LIN {X 0,Y 270.05,Z 181.094,A -85,B 0,C 180,E1 -19060.447,E2 -19060.447} C_VEL
LIN {X 0,Y 266.904,Z 176.821,A -85,B 0,C 180,E1 -19061.814,E2 -19061.814} C_VEL
LIN {X 0,Y 264.347,Z 175.041,A -85,B 0,C 180,E1 -19062.905,E2 -19062.905} C_VEL
LIN {X 0,Y 256.649,Z 172.883,A -85,B 0,C 180,E1 -19066.441,E2 -19066.441} C_VEL
LIN {X 0,Y 254.506,Z 171.313,A -85,B 0,C 180,E1 -19067.626,E2 -19067.626} C_VEL
LIN {X 0,Y 253.888,Z 170.514,A -85,B 0,C 180,E1 -19068.008,E2 -19068.008} C_VEL
LIN {X 0,Y 252.108,Z 167.577,A -85,B 0,C 180,E1 -19069.204,E2 -19069.204} C_VEL
LIN {X 0,Y 249.588,Z 165.512,A -85,B 0,C 180,E1 -19070.909,E2 -19070.909} C_VEL
LIN {X 0,Y 247.997,Z 162.813,A -85,B 0,C 180,E1 -19072.212,E2 -19072.212} C_VEL
LIN {X 0,Y 247.745,Z 162.046,A -85,B 0,C 180,E1 -19072.46,E2 -19072.46} C_VEL
LIN {X 0,Y 244.192,Z 159.968,A -85,B 0,C 180,E1 -19075.46,E2 -19075.46} C_VEL
LIN {X 0,Y 242.872,Z 157.671,A -85,B 0,C 180,E1 -19076.993,E2 -19076.993} C_VEL
LIN {X 0,Y 242.522,Z 155.89,A -85,B 0,C 180,E1 -19077.716,E2 -19077.716} C_VEL
LIN {X 0,Y 242.691,Z 155.88,A -85,B 0,C 180,E1 -19079.999,E2 -19079.999} C_VEL
LIN {X 0,Y 242.635,Z 155.875,A -85,B 0,C 180,E1 -19081.659,E2 -19081.659} C_VEL
LIN {X 0,Y 242.4,Z 155.913,A -85,B 0,C 180,E1 -19086.659,E2 -19086.659} C_VEL
LIN {X 0,Y 242.265,Z 155.926,A -85,B 0,C 180,E1 -19090.023,E2 -19090.023} C_VEL
LIN {X 0,Y 242.166,Z 155.938,A -85,B 0,C 180,E1 -19095.14,E2 -19095.14} C_VEL
LIN {X 0,Y 242.075,Z 155.945,A -85,B 0,C 180,E1 -19099.669,E2 -19099.669} C_VEL
LIN {X 0,Y 242.299,Z 157.093,A -85,B 0,C 180,E1 -19100.991,E2 -19100.991} C_VEL
LIN {X 0,Y 243.437,Z 159.421,A -85,B 0,C 180,E1 -19102.448,E2 -19102.448} C_VEL
LIN {X 0,Y 246.039,Z 161.798,A -85,B 0,C 180,E1 -19104.918,E2 -19104.918} C_VEL
LIN {X 0,Y 248.946,Z 165.199,A -85,B 0,C 180,E1 -19107.306,E2 -19107.306} C_VEL
LIN {X 0,Y 252.346,Z 169.692,A -85,B 0,C 180,E1 -19109.752,E2 -19109.752} C_VEL
LIN {X 0,Y 253.782,Z 171.342,A -85,B 0,C 180,E1 -19110.657,E2 -19110.657} C_VEL
LIN {X 0,Y 258.589,Z 177.663,A -85,B 0,C 180,E1 -19113.449,E2 -19113.449} C_VEL
LIN {X 0,Y 262.502,Z 183.277,A -85,B 0,C 180,E1 -19115.489,E2 -19115.489} C_VEL
LIN {X 0,Y 268.007,Z 191.52,A -85,B 0,C 180,E1 -19118.035,E2 -19118.035} C_VEL
LIN {X 0,Y 273.834,Z 200.761,A -85,B 0,C 180,E1 -19120.447,E2 -19120.447} C_VEL
LIN {X 0,Y 279.53,Z 210.74,A -85,B 0,C 180,E1 -19122.615,E2 -19122.615} C_VEL
LIN {X 0,Y 285.287,Z 221.644,A -85,B 0,C 180,E1 -19124.619,E2 -19124.619} C_VEL
LIN {X 0,Y 291.028,Z 234.204,A -85,B 0,C 180,E1 -19126.505,E2 -19126.505} C_VEL
LIN {X 0,Y 291.336,Z 235.609,A -85,B 0,C 180,E1 -19126.631,E2 -19126.631} C_VEL
LIN {X 0,Y 285.753,Z 326.096,A -85,B 0,C 180,E1 -19128.86,E2 -19128.86} C_VEL
LIN {X 0,Y 283.787,Z 341.992,A -85,B 0,C 180,E1 -19129.453,E2 -19129.453} C_VEL
LIN {X 0,Y 281.088,Z 357.105,A -85,B 0,C 180,E1 -19130.273,E2 -19130.273} C_VEL
LIN {X 0,Y 278.009,Z 370.686,A -85,B 0,C 180,E1 -19131.269,E2 -19131.269} C_VEL
LIN {X 0,Y 274.119,Z 385.222,A -85,B 0,C 180,E1 -19132.661,E2 -19132.661} C_VEL
LIN {X 0,Y 270.67,Z 396.438,A -85,B 0,C 180,E1 -19134.023,E2 -19134.023} C_VEL
LIN {X 0,Y 266.245,Z 409.051,A -85,B 0,C 180,E1 -19135.88,E2 -19135.88} C_VEL
LIN {X 0,Y 261.748,Z 420.548,A -85,B 0,C 180,E1 -19137.975,E2 -19137.975} C_VEL
LIN {X 0,Y 257.041,Z 431.736,A -85,B 0,C 180,E1 -19140.518,E2 -19140.518} C_VEL
LIN {X 0,Y 253.709,Z 439.245,A -85,B 0,C 180,E1 -19142.582,E2 -19142.582} C_VEL
LIN {X 0,Y 249.879,Z 447.882,A -85,B 0,C 180,E1 -19145.491,E2 -19145.491} C_VEL
LIN {X 0,Y 246.86,Z 454.558,A -85,B 0,C 180,E1 -19148.279,E2 -19148.279} C_VEL
LIN {X 0,Y 244,Z 460.761,A -85,B 0,C 180,E1 -19151.529,E2 -19151.529} C_VEL
LIN {X 0,Y 242.026,Z 465.605,A -85,B 0,C 180,E1 -19154.851,E2 -19154.851} C_VEL
LIN {X 0,Y 240.671,Z 469.21,A -85,B 0,C 180,E1 -19158.206,E2 -19158.206} C_VEL
LIN {X 0,Y 239.979,Z 471.652,A -85,B 0,C 180,E1 -19161.581,E2 -19161.581} C_VEL
LIN {X 0,Y 239.733,Z 473.016,A -85,B 0,C 180,E1 -19165.368,E2 -19165.368} C_VEL
LIN {X 0,Y 239.826,Z 473.079,A -85,B 0,C 180,E1 -19168.321,E2 -19168.321} C_VEL
LIN {X 0,Y 239.912,Z 472.714,A -85,B 0,C 180,E1 -19170.001,E2 -19170.001} C_VEL
LIN {X 0,Y 239.783,Z 471.099,A -85,B 0,C 180,E1 -19173.361,E2 -19173.361} C_VEL
LIN {X 0,Y 239.876,Z 468.281,A -85,B 0,C 180,E1 -19176.731,E2 -19176.731} C_VEL
LIN {X 0,Y 240.194,Z 464.175,A -85,B 0,C 180,E1 -19180.112,E2 -19180.112} C_VEL
LIN {X 0,Y 241.031,Z 458.673,A -85,B 0,C 180,E1 -19183.49,E2 -19183.49} C_VEL
LIN {X 0,Y 242.441,Z 451.405,A -85,B 0,C 180,E1 -19186.94,E2 -19186.94} C_VEL
LIN {X 0,Y 244.164,Z 444.018,A -85,B 0,C 180,E1 -19189.769,E2 -19189.769} C_VEL
LIN {X 0,Y 246.564,Z 434.858,A -85,B 0,C 180,E1 -19192.632,E2 -19192.632} C_VEL
LIN {X 0,Y 249.211,Z 424.133,A -85,B 0,C 180,E1 -19195.381,E2 -19195.381} C_VEL
LIN {X 0,Y 252.238,Z 412.368,A -85,B 0,C 180,E1 -19197.821,E2 -19197.821} C_VEL
LIN {X 0,Y 255.134,Z 399.787,A -85,B 0,C 180,E1 -19199.953,E2 -19199.953} C_VEL
LIN {X 0,Y 257.953,Z 387.419,A -85,B 0,C 180,E1 -19201.634,E2 -19201.634} C_VEL
LIN {X 0,Y 260.774,Z 372.915,A -85,B 0,C 180,E1 -19203.222,E2 -19203.222} C_VEL
LIN {X 0,Y 263.081,Z 358.225,A -85,B 0,C 180,E1 -19204.473,E2 -19204.473} C_VEL
LIN {X 0,Y 265.181,Z 342.628,A -85,B 0,C 180,E1 -19205.434,E2 -19205.434} C_VEL
LIN {X 0,Y 266.583,Z 327.14,A -85,B 0,C 180,E1 -19206.091,E2 -19206.091} C_VEL
LIN {X 0,Y 271.19,Z 222.807,A -85,B 0,C 180,E1 -19208.824,E2 -19208.824} C_VEL
LIN {X 0,Y 270.291,Z 218.299,A -85,B 0,C 180,E1 -19209.091,E2 -19209.091} C_VEL
LIN {X 0,Y 263.458,Z 201.272,A -85,B 0,C 180,E1 -19210.628,E2 -19210.628} C_VEL
LIN {X 0,Y 255.801,Z 184.265,A -85,B 0,C 180,E1 -19212.402,E2 -19212.402} C_VEL
LIN {X 0,Y 248.125,Z 169.408,A -85,B 0,C 180,E1 -19214.242,E2 -19214.242} C_VEL
LIN {X 0,Y 243.223,Z 160.405,A -85,B 0,C 180,E1 -19215.517,E2 -19215.517} C_VEL
LIN {X 0,Y 241.97,Z 155.973,A -85,B 0,C 180,E1 -19217.349,E2 -19217.349} C_VEL
LIN {X 0,Y 241.997,Z 155.954,A -85,B 0,C 180,E1 -19221.641,E2 -19221.641} C_VEL
LIN {X 0,Y 241.989,Z 155.963,A -85,B 0,C 180,E1 -19224.49,E2 -19224.49} C_VEL
LIN {X 0,Y 241.955,Z 155.97,A -85,B 0,C 180,E1 -19228.478,E2 -19228.478} C_VEL
LIN {X 0,Y 241.97,Z 155.934,A -85,B 0,C 180,E1 -19232.309,E2 -19232.309} C_VEL
LIN {X 0,Y 242.028,Z 155.96,A -85,B 0,C 180,E1 -19236.014,E2 -19236.014} C_VEL
LIN {X 0,Y 242.025,Z 155.958,A -85,B 0,C 180,E1 -19239.607,E2 -19239.607} C_VEL
LIN {X 0,Y 242.131,Z 155.938,A -85,B 0,C 180,E1 -19243.308,E2 -19243.308} C_VEL
LIN {X 0,Y 242.172,Z 155.936,A -85,B 0,C 180,E1 -19248.28,E2 -19248.28} C_VEL
LIN {X 0,Y 242.376,Z 155.912,A -85,B 0,C 180,E1 -19251.664,E2 -19251.664} C_VEL
LIN {X 0,Y 242.401,Z 155.911,A -85,B 0,C 180,E1 -19253.341,E2 -19253.341} C_VEL
LIN {X 0,Y 242.621,Z 155.851,A -85,B 0,C 180,E1 -19258.341,E2 -19258.341} C_VEL
LIN {X 0,Y 242.619,Z 155.864,A -85,B 0,C 180,E1 -19261.661,E2 -19261.661} C_VEL
LIN {X 0,Y 242.4,Z 155.901,A -85,B 0,C 180,E1 -19266.66,E2 -19266.66} C_VEL
LIN {X 0,Y 242.264,Z 155.888,A -85,B 0,C 180,E1 -19270.025,E2 -19270.025} C_VEL
LIN {X 0,Y 242.106,Z 155.951,A -85,B 0,C 180,E1 -19275.145,E2 -19275.145} C_VEL
LIN {X 0,Y 242.013,Z 155.961,A -85,B 0,C 180,E1 -19278.63,E2 -19278.63} C_VEL
LIN {X 0,Y 241.975,Z 155.958,A -85,B 0,C 180,E1 -19282.184,E2 -19282.184} C_VEL
LIN {X 0,Y 241.991,Z 155.962,A -85,B 0,C 180,E1 -19285.827,E2 -19285.827} C_VEL
LIN {X 0,Y 241.967,Z 155.928,A -85,B 0,C 180,E1 -19289.59,E2 -19289.59} C_VEL
LIN {X 0,Y 241.983,Z 155.967,A -85,B 0,C 180,E1 -19293.493,E2 -19293.493} C_VEL
LIN {X 0,Y 241.988,Z 155.932,A -85,B 0,C 180,E1 -19297.583,E2 -19297.583} C_VEL
LIN {X 0,Y 241.923,Z 155.974,A -85,B 0,C 180,E1 -19301.927,E2 -19301.927} C_VEL
LIN {X 0,Y 241.904,Z 155.951,A -85,B 0,C 180,E1 -19306.58,E2 -19306.58} C_VEL
LIN {X 0,Y 241.934,Z 155.969,A -85,B 0,C 180,E1 -19310.276,E2 -19310.276} C_VEL
LIN {X 0,Y 241.978,Z 155.966,A -85,B 0,C 180,E1 -19314.487,E2 -19314.487} C_VEL
LIN {X 0,Y 241.958,Z 155.961,A -85,B 0,C 180,E1 -19318.476,E2 -19318.476} C_VEL
LIN {X 0,Y 241.969,Z 155.963,A -85,B 0,C 180,E1 -19322.307,E2 -19322.307} C_VEL
LIN {X 0,Y 241.999,Z 156.029,A -85,B 0,C 180,E1 -19323.589,E2 -19323.589} C_VEL
LIN {X 0,Y 242.921,Z 158.683,A -85,B 0,C 180,E1 -19323.869,E2 -19323.869} C_VEL
LIN {X 0,Y 244.718,Z 161.076,A -85,B 0,C 180,E1 -19324.3,E2 -19324.3} C_VEL
LIN {X 0,Y 256.472,Z 180.366,A -85,B 0,C 180,E1 -19327.043,E2 -19327.043} C_VEL
LIN {X 0,Y 262.923,Z 192.515,A -85,B 0,C 180,E1 -19328.47,E2 -19328.47} C_VEL
LIN {X 0,Y 269.632,Z 208.086,A -85,B 0,C 180,E1 -19329.962,E2 -19329.962} C_VEL
LIN {X 0,Y 271.569,Z 213.034,A -85,B 0,C 180,E1 -19330.389,E2 -19330.389} C_VEL
LIN {X 0,Y 266.876,Z 314.239,A -85,B 0,C 180,E1 -19333.013,E2 -19333.013} C_VEL
LIN {X 0,Y 265.518,Z 330.347,A -85,B 0,C 180,E1 -19333.715,E2 -19333.715} C_VEL
LIN {X 0,Y 263.826,Z 344.934,A -85,B 0,C 180,E1 -19334.649,E2 -19334.649} C_VEL
LIN {X 0,Y 261.727,Z 358.741,A -85,B 0,C 180,E1 -19335.816,E2 -19335.816} C_VEL
LIN {X 0,Y 259.363,Z 371.908,A -85,B 0,C 180,E1 -19337.229,E2 -19337.229} C_VEL
LIN {X 0,Y 256.641,Z 384.864,A -85,B 0,C 180,E1 -19338.948,E2 -19338.948} C_VEL
LIN {X 0,Y 253.902,Z 396.522,A -85,B 0,C 180,E1 -19340.841,E2 -19340.841} C_VEL
LIN {X 0,Y 251.026,Z 408.225,A -85,B 0,C 180,E1 -19343.166,E2 -19343.166} C_VEL
LIN {X 0,Y 248.456,Z 418.09,A -85,B 0,C 180,E1 -19345.538,E2 -19345.538} C_VEL
LIN {X 0,Y 246.001,Z 427.734,A -85,B 0,C 180,E1 -19348.362,E2 -19348.362} C_VEL
LIN {X 0,Y 243.924,Z 435.785,A -85,B 0,C 180,E1 -19351.238,E2 -19351.238} C_VEL
LIN {X 0,Y 242.335,Z 442.479,A -85,B 0,C 180,E1 -19354.157,E2 -19354.157} C_VEL
LIN {X 0,Y 241.036,Z 448.623,A -85,B 0,C 180,E1 -19357.533,E2 -19357.533} C_VEL
LIN {X 0,Y 240.172,Z 453.365,A -85,B 0,C 180,E1 -19360.964,E2 -19360.964} C_VEL
LIN {X 0,Y 239.642,Z 456.898,A -85,B 0,C 180,E1 -19364.578,E2 -19364.578} C_VEL
LIN {X 0,Y 239.493,Z 458.496,A -85,B 0,C 180,E1 -19367.064,E2 -19367.064} C_VEL
LIN {X 0,Y 239.492,Z 459.74,A -85,B 0,C 180,E1 -19370.618,E2 -19370.618} C_VEL
LIN {X 0,Y 239.842,Z 459.722,A -85,B 0,C 180,E1 -19374.219,E2 -19374.219} C_VEL
LIN {X 0,Y 240.587,Z 458.394,A -85,B 0,C 180,E1 -19377.864,E2 -19377.864} C_VEL
LIN {X 0,Y 241.902,Z 455.693,A -85,B 0,C 180,E1 -19381.53,E2 -19381.53} C_VEL
LIN {X 0,Y 243.937,Z 451.533,A -85,B 0,C 180,E1 -19385.184,E2 -19385.184} C_VEL
LIN {X 0,Y 246.746,Z 445.781,A -85,B 0,C 180,E1 -19388.801,E2 -19388.801} C_VEL
LIN {X 0,Y 249.894,Z 439.307,A -85,B 0,C 180,E1 -19391.908,E2 -19391.908} C_VEL
LIN {X 0,Y 253.681,Z 431.274,A -85,B 0,C 180,E1 -19394.946,E2 -19394.946} C_VEL
LIN {X 0,Y 258.142,Z 421.415,A -85,B 0,C 180,E1 -19397.892,E2 -19397.892} C_VEL
LIN {X 0,Y 262.699,Z 410.7,A -85,B 0,C 180,E1 -19400.441,E2 -19400.441} C_VEL
LIN {X 0,Y 267.081,Z 399.355,A -85,B 0,C 180,E1 -19402.624,E2 -19402.624} C_VEL
LIN {X 0,Y 271.14,Z 387.871,A -85,B 0,C 180,E1 -19404.414,E2 -19404.414} C_VEL
LIN {X 0,Y 275.252,Z 374.612,A -85,B 0,C 180,E1 -19406.081,E2 -19406.081} C_VEL
LIN {X 0,Y 278.751,Z 360.969,A -85,B 0,C 180,E1 -19407.462,E2 -19407.462} C_VEL
LIN {X 0,Y 282.029,Z 345.738,A -85,B 0,C 180,E1 -19408.632,E2 -19408.632} C_VEL
LIN {X 0,Y 284.295,Z 332.001,A -85,B 0,C 180,E1 -19409.426,E2 -19409.426} C_VEL
LIN {X 0,Y 286.217,Z 316.146,A -85,B 0,C 180,E1 -19410.059,E2 -19410.059} C_VEL
LIN {X 0,Y 291.678,Z 227.342,A -85,B 0,C 180,E1 -19412.267,E2 -19412.267} C_VEL
LIN {X 0,Y 286.52,Z 216.955,A -85,B 0,C 180,E1 -19413.922,E2 -19413.922} C_VEL
LIN {X 0,Y 280.857,Z 206.853,A -85,B 0,C 180,E1 -19415.843,E2 -19415.843} C_VEL
LIN {X 0,Y 276.3,Z 199.31,A -85,B 0,C 180,E1 -19417.519,E2 -19417.519} C_VEL
LIN {X 0,Y 270.649,Z 191.335,A -85,B 0,C 180,E1 -19419.718,E2 -19419.718} C_VEL
LIN {X 0,Y 267.391,Z 187.043,A -85,B 0,C 180,E1 -19421.082,E2 -19421.082} C_VEL
LIN {X 0,Y 264.021,Z 182.609,A -85,B 0,C 180,E1 -19422.595,E2 -19422.595} C_VEL
LIN {X 0,Y 261.176,Z 178.839,A -85,B 0,C 180,E1 -19423.994,E2 -19423.994} C_VEL
LIN {X 0,Y 257.612,Z 174.63,A -85,B 0,C 180,E1 -19425.862,E2 -19425.862} C_VEL
LIN {X 0,Y 256.541,Z 173.01,A -85,B 0,C 180,E1 -19426.483,E2 -19426.483} C_VEL
LIN {X 0,Y 253.888,Z 170.514,A -85,B 0,C 180,E1 -19428.008,E2 -19428.008} C_VEL
LIN {X 0,Y 251.988,Z 168.678,A -85,B 0,C 180,E1 -19429.196,E2 -19429.196} C_VEL
LIN {X 0,Y 249.958,Z 168.052,A -85,B 0,C 180,E1 -19430.459,E2 -19430.459} C_VEL
LIN {X 0,Y 244.872,Z 168.118,A -85,B 0,C 180,E1 -19434,E2 -19434} C_VEL
LIN {X 0,Y 243.834,Z 167.609,A -85,B 0,C 180,E1 -19434.905,E2 -19434.905} C_VEL
LIN {X 0,Y 241.974,Z 165.418,A -85,B 0,C 180,E1 -19436.878,E2 -19436.878} C_VEL
LIN {X 0,Y 240.963,Z 162.777,A -85,B 0,C 180,E1 -19438.328,E2 -19438.328} C_VEL
LIN {X 0,Y 236.581,Z 159.994,A -85,B 0,C 180,E1 -19448.541,E2 -19448.541} C_VEL
LIN {X 0,Y 237.634,Z 161.379,A -85,B 0,C 180,E1 -19454.997,E2 -19454.997} C_VEL
LIN {X 0,Y 240.519,Z 163.072,A -85,B 0,C 180,E1 -19459.857,E2 -19459.857} C_VEL
LIN {X 0,Y 241.092,Z 164.194,A -85,B 0,C 180,E1 -19460.684,E2 -19460.684} C_VEL
LIN {X 0,Y 242.46,Z 166.569,A -85,B 0,C 180,E1 -19462.408,E2 -19462.408} C_VEL
LIN {X 0,Y 244.723,Z 168.674,A -85,B 0,C 180,E1 -19464.604,E2 -19464.604} C_VEL
LIN {X 0,Y 247.713,Z 172.251,A -85,B 0,C 180,E1 -19467.118,E2 -19467.118} C_VEL
LIN {X 0,Y 250.494,Z 176.134,A -85,B 0,C 180,E1 -19469.197,E2 -19469.197} C_VEL
LIN {X 0,Y 251.866,Z 177.723,A -85,B 0,C 180,E1 -19470.094,E2 -19470.094} C_VEL
LIN {X 0,Y 257.149,Z 185.048,A -85,B 0,C 180,E1 -19473.266,E2 -19473.266} C_VEL
LIN {X 0,Y 261.114,Z 190.954,A -85,B 0,C 180,E1 -19475.371,E2 -19475.371} C_VEL
LIN {X 0,Y 265.433,Z 197.515,A -85,B 0,C 180,E1 -19477.424,E2 -19477.424} C_VEL
LIN {X 0,Y 271.29,Z 207.09,A -85,B 0,C 180,E1 -19479.938,E2 -19479.938} C_VEL
LIN {X 0,Y 277.493,Z 218.235,A -85,B 0,C 180,E1 -19482.363,E2 -19482.363} C_VEL
LIN {X 0,Y 282.654,Z 228.654,A -85,B 0,C 180,E1 -19484.231,E2 -19484.231} C_VEL
LIN {X 0,Y 286.593,Z 237.467,A -85,B 0,C 180,E1 -19485.579,E2 -19485.579} C_VEL
LIN {X 0,Y 280.938,Z 326.652,A -85,B 0,C 180,E1 -19487.815,E2 -19487.815} C_VEL
LIN {X 0,Y 278.906,Z 342.252,A -85,B 0,C 180,E1 -19488.409,E2 -19488.409} C_VEL
LIN {X 0,Y 275.999,Z 357.801,A -85,B 0,C 180,E1 -19489.269,E2 -19489.269} C_VEL
LIN {X 0,Y 273.075,Z 370.282,A -85,B 0,C 180,E1 -19490.194,E2 -19490.194} C_VEL
LIN {X 0,Y 268.999,Z 385.006,A -85,B 0,C 180,E1 -19491.609,E2 -19491.609} C_VEL
LIN {X 0,Y 265.419,Z 396.114,A -85,B 0,C 180,E1 -19492.959,E2 -19492.959} C_VEL
LIN {X 0,Y 260.837,Z 408.746,A -85,B 0,C 180,E1 -19494.836,E2 -19494.836} C_VEL
LIN {X 0,Y 256.529,Z 419.379,A -85,B 0,C 180,E1 -19496.775,E2 -19496.775} C_VEL
LIN {X 0,Y 252.236,Z 429.258,A -85,B 0,C 180,E1 -19498.972,E2 -19498.972} C_VEL
LIN {X 0,Y 247.788,Z 438.738,A -85,B 0,C 180,E1 -19501.551,E2 -19501.551} C_VEL
LIN {X 0,Y 243.972,Z 447.08,A -85,B 0,C 180,E1 -19504.4,E2 -19504.4} C_VEL
LIN {X 0,Y 240.238,Z 454.728,A -85,B 0,C 180,E1 -19507.648,E2 -19507.648} C_VEL
LIN {X 0,Y 237.243,Z 460.853,A -85,B 0,C 180,E1 -19510.983,E2 -19510.983} C_VEL
LIN {X 0,Y 235.103,Z 465.624,A -85,B 0,C 180,E1 -19514.393,E2 -19514.393} C_VEL
LIN {X 0,Y 233.667,Z 469.158,A -85,B 0,C 180,E1 -19517.847,E2 -19517.847} C_VEL
LIN {X 0,Y 232.918,Z 471.531,A -85,B 0,C 180,E1 -19521.323,E2 -19521.323} C_VEL
LIN {X 0,Y 232.644,Z 472.783,A -85,B 0,C 180,E1 -19524.801,E2 -19524.801} C_VEL
LIN {X 0,Y 232.737,Z 472.864,A -85,B 0,C 180,E1 -19528.27,E2 -19528.27} C_VEL
LIN {X 0,Y 232.821,Z 472.468,A -85,B 0,C 180,E1 -19530.001,E2 -19530.001} C_VEL
LIN {X 0,Y 232.693,Z 470.79,A -85,B 0,C 180,E1 -19533.464,E2 -19533.464} C_VEL
LIN {X 0,Y 232.792,Z 467.905,A -85,B 0,C 180,E1 -19536.937,E2 -19536.937} C_VEL
LIN {X 0,Y 233.139,Z 463.729,A -85,B 0,C 180,E1 -19540.421,E2 -19540.421} C_VEL
LIN {X 0,Y 234.062,Z 458.154,A -85,B 0,C 180,E1 -19543.9,E2 -19543.9} C_VEL
LIN {X 0,Y 235.539,Z 451.013,A -85,B 0,C 180,E1 -19547.361,E2 -19547.361} C_VEL
LIN {X 0,Y 237.393,Z 443.346,A -85,B 0,C 180,E1 -19550.357,E2 -19550.357} C_VEL
LIN {X 0,Y 239.93,Z 434.093,A -85,B 0,C 180,E1 -19553.294,E2 -19553.294} C_VEL
LIN {X 0,Y 242.816,Z 422.819,A -85,B 0,C 180,E1 -19556.201,E2 -19556.201} C_VEL
LIN {X 0,Y 245.869,Z 411.284,A -85,B 0,C 180,E1 -19558.607,E2 -19558.607} C_VEL
LIN {X 0,Y 248.916,Z 398.506,A -85,B 0,C 180,E1 -19560.781,E2 -19560.781} C_VEL
LIN {X 0,Y 251.821,Z 385.956,A -85,B 0,C 180,E1 -19562.497,E2 -19562.497} C_VEL
LIN {X 0,Y 254.454,Z 372.935,A -85,B 0,C 180,E1 -19563.931,E2 -19563.931} C_VEL
LIN {X 0,Y 256.812,Z 358.412,A -85,B 0,C 180,E1 -19565.199,E2 -19565.199} C_VEL
LIN {X 0,Y 258.974,Z 342.993,A -85,B 0,C 180,E1 -19566.176,E2 -19566.176} C_VEL
LIN {X 0,Y 260.407,Z 327.797,A -85,B 0,C 180,E1 -19566.846,E2 -19566.846} C_VEL
LIN {X 0,Y 265.233,Z 224.118,A -85,B 0,C 180,E1 -19569.612,E2 -19569.612} C_VEL
LIN {X 0,Y 264.413,Z 220.374,A -85,B 0,C 180,E1 -19569.853,E2 -19569.853} C_VEL
LIN {X 0,Y 256.732,Z 201.426,A -85,B 0,C 180,E1 -19571.658,E2 -19571.658} C_VEL
LIN {X 0,Y 249.37,Z 185.374,A -85,B 0,C 180,E1 -19573.436,E2 -19573.436} C_VEL
LIN {X 0,Y 242.22,Z 171.766,A -85,B 0,C 180,E1 -19575.234,E2 -19575.234} C_VEL
LIN {X 0,Y 235.916,Z 160.21,A -85,B 0,C 180,E1 -19576.945,E2 -19576.945} C_VEL
LIN {X 0,Y 234.882,Z 156.856,A -85,B 0,C 180,E1 -19578.422,E2 -19578.422} C_VEL
LIN {X 0,Y 234.92,Z 156.834,A -85,B 0,C 180,E1 -19581.08,E2 -19581.08} C_VEL
LIN {X 0,Y 234.932,Z 156.845,A -85,B 0,C 180,E1 -19585.363,E2 -19585.363} C_VEL
LIN {X 0,Y 234.901,Z 156.847,A -85,B 0,C 180,E1 -19589.429,E2 -19589.429} C_VEL
LIN {X 0,Y 234.971,Z 156.814,A -85,B 0,C 180,E1 -19593.808,E2 -19593.808} C_VEL
LIN {X 0,Y 234.993,Z 156.828,A -85,B 0,C 180,E1 -19598.969,E2 -19598.969} C_VEL
LIN {X 0,Y 235.067,Z 156.818,A -85,B 0,C 180,E1 -19603.087,E2 -19603.087} C_VEL
LIN {X 0,Y 235.104,Z 156.815,A -85,B 0,C 180,E1 -19607.922,E2 -19607.922} C_VEL
LIN {X 0,Y 235.315,Z 156.793,A -85,B 0,C 180,E1 -19611.412,E2 -19611.412} C_VEL
LIN {X 0,Y 235.352,Z 156.787,A -85,B 0,C 180,E1 -19613.141,E2 -19613.141} C_VEL
LIN {X 0,Y 235.58,Z 156.727,A -85,B 0,C 180,E1 -19618.291,E2 -19618.291} C_VEL
LIN {X 0,Y 235.578,Z 156.741,A -85,B 0,C 180,E1 -19621.71,E2 -19621.71} C_VEL
LIN {X 0,Y 235.351,Z 156.774,A -85,B 0,C 180,E1 -19626.861,E2 -19626.861} C_VEL
LIN {X 0,Y 235.187,Z 156.77,A -85,B 0,C 180,E1 -19630.329,E2 -19630.329} C_VEL
LIN {X 0,Y 235.044,Z 156.827,A -85,B 0,C 180,E1 -19635.612,E2 -19635.612} C_VEL
LIN {X 0,Y 234.956,Z 156.841,A -85,B 0,C 180,E1 -19639.211,E2 -19639.211} C_VEL
LIN {X 0,Y 234.919,Z 156.839,A -85,B 0,C 180,E1 -19642.888,E2 -19642.888} C_VEL
LIN {X 0,Y 234.926,Z 156.832,A -85,B 0,C 180,E1 -19646.664,E2 -19646.664} C_VEL
LIN {X 0,Y 234.899,Z 156.813,A -85,B 0,C 180,E1 -19650.573,E2 -19650.573} C_VEL
LIN {X 0,Y 234.927,Z 156.845,A -85,B 0,C 180,E1 -19654.639,E2 -19654.639} C_VEL
LIN {X 0,Y 234.917,Z 156.813,A -85,B 0,C 180,E1 -19658.935,E2 -19658.935} C_VEL
LIN {X 0,Y 234.866,Z 156.848,A -85,B 0,C 180,E1 -19663.492,E2 -19663.492} C_VEL
LIN {X 0,Y 234.857,Z 156.828,A -85,B 0,C 180,E1 -19666.506,E2 -19666.506} C_VEL
LIN {X 0,Y 234.923,Z 156.833,A -85,B 0,C 180,E1 -19671.078,E2 -19671.078} C_VEL
LIN {X 0,Y 234.927,Z 156.847,A -85,B 0,C 180,E1 -19675.36,E2 -19675.36} C_VEL
LIN {X 0,Y 234.904,Z 156.853,A -85,B 0,C 180,E1 -19679.427,E2 -19679.427} C_VEL
LIN {X 0,Y 234.937,Z 156.838,A -85,B 0,C 180,E1 -19682.195,E2 -19682.195} C_VEL
LIN {X 0,Y 235.938,Z 159.689,A -85,B 0,C 180,E1 -19682.53,E2 -19682.53} C_VEL
LIN {X 0,Y 237.799,Z 162.132,A -85,B 0,C 180,E1 -19683.003,E2 -19683.003} C_VEL
LIN {X 0,Y 246.976,Z 176.903,A -85,B 0,C 180,E1 -19685.309,E2 -19685.309} C_VEL
LIN {X 0,Y 254.136,Z 189.258,A -85,B 0,C 180,E1 -19686.979,E2 -19686.979} C_VEL
LIN {X 0,Y 258.788,Z 198.574,A -85,B 0,C 180,E1 -19688.04,E2 -19688.04} C_VEL
LIN {X 0,Y 265.578,Z 214.964,A -85,B 0,C 180,E1 -19689.609,E2 -19689.609} C_VEL
LIN {X 0,Y 260.744,Z 314.885,A -85,B 0,C 180,E1 -19692.246,E2 -19692.246} C_VEL
LIN {X 0,Y 259.332,Z 330.805,A -85,B 0,C 180,E1 -19692.96,E2 -19692.96} C_VEL
LIN {X 0,Y 257.524,Z 345.902,A -85,B 0,C 180,E1 -19693.959,E2 -19693.959} C_VEL
LIN {X 0,Y 255.157,Z 360.523,A -85,B 0,C 180,E1 -19695.239,E2 -19695.239} C_VEL
LIN {X 0,Y 252.495,Z 374.776,A -85,B 0,C 180,E1 -19696.861,E2 -19696.861} C_VEL
LIN {X 0,Y 249.667,Z 387.4,A -85,B 0,C 180,E1 -19698.635,E2 -19698.635} C_VEL
LIN {X 0,Y 246.618,Z 399.734,A -85,B 0,C 180,E1 -19700.775,E2 -19700.775} C_VEL
LIN {X 0,Y 243.513,Z 411.782,A -85,B 0,C 180,E1 -19703.37,E2 -19703.37} C_VEL
LIN {X 0,Y 240.949,Z 421.166,A -85,B 0,C 180,E1 -19705.818,E2 -19705.818} C_VEL
LIN {X 0,Y 238.518,Z 430.331,A -85,B 0,C 180,E1 -19708.733,E2 -19708.733} C_VEL
LIN {X 0,Y 236.493,Z 437.957,A -85,B 0,C 180,E1 -19711.702,E2 -19711.702} C_VEL
LIN {X 0,Y 234.793,Z 445.088,A -85,B 0,C 180,E1 -19715.151,E2 -19715.151} C_VEL
LIN {X 0,Y 233.602,Z 450.702,A -85,B 0,C 180,E1 -19718.651,E2 -19718.651} C_VEL
LIN {X 0,Y 232.826,Z 454.939,A -85,B 0,C 180,E1 -19722.198,E2 -19722.198} C_VEL
LIN {X 0,Y 232.427,Z 457.891,A -85,B 0,C 180,E1 -19725.791,E2 -19725.791} C_VEL
LIN {X 0,Y 232.364,Z 459.599,A -85,B 0,C 180,E1 -19729.432,E2 -19729.432} C_VEL
LIN {X 0,Y 232.561,Z 460.062,A -85,B 0,C 180,E1 -19733.132,E2 -19733.132} C_VEL
LIN {X 0,Y 233.2,Z 459.239,A -85,B 0,C 180,E1 -19736.875,E2 -19736.875} C_VEL
LIN {X 0,Y 234.434,Z 457.076,A -85,B 0,C 180,E1 -19740.639,E2 -19740.639} C_VEL
LIN {X 0,Y 236.295,Z 453.486,A -85,B 0,C 180,E1 -19744.409,E2 -19744.409} C_VEL
LIN {X 0,Y 239.011,Z 448.36,A -85,B 0,C 180,E1 -19748.133,E2 -19748.133} C_VEL
LIN {X 0,Y 241.528,Z 443.525,A -85,B 0,C 180,E1 -19750.838,E2 -19750.838} C_VEL
LIN {X 0,Y 244.607,Z 437.421,A -85,B 0,C 180,E1 -19753.595,E2 -19753.595} C_VEL
LIN {X 0,Y 248.8,Z 428.94,A -85,B 0,C 180,E1 -19756.666,E2 -19756.666} C_VEL
LIN {X 0,Y 252.948,Z 420.173,A -85,B 0,C 180,E1 -19759.21,E2 -19759.21} C_VEL
LIN {X 0,Y 257.636,Z 409.469,A -85,B 0,C 180,E1 -19761.725,E2 -19761.725} C_VEL
LIN {X 0,Y 262.414,Z 397.448,A -85,B 0,C 180,E1 -19763.986,E2 -19763.986} C_VEL
LIN {X 0,Y 266.674,Z 385.585,A -85,B 0,C 180,E1 -19765.777,E2 -19765.777} C_VEL
LIN {X 0,Y 270.928,Z 371.743,A -85,B 0,C 180,E1 -19767.463,E2 -19767.463} C_VEL
LIN {X 0,Y 274.264,Z 359.022,A -85,B 0,C 180,E1 -19768.691,E2 -19768.691} C_VEL
LIN {X 0,Y 277.216,Z 345.478,A -85,B 0,C 180,E1 -19769.717,E2 -19769.717} C_VEL
LIN {X 0,Y 279.621,Z 331.257,A -85,B 0,C 180,E1 -19770.534,E2 -19770.534} C_VEL
LIN {X 0,Y 281.563,Z 315.4,A -85,B 0,C 180,E1 -19771.146,E2 -19771.146} C_VEL
LIN {X 0,Y 286.987,Z 230.143,A -85,B 0,C 180,E1 -19773.276,E2 -19773.276} C_VEL
LIN {X 0,Y 281.02,Z 218.276,A -85,B 0,C 180,E1 -19775.3,E2 -19775.3} C_VEL
LIN {X 0,Y 273.795,Z 205.579,A -85,B 0,C 180,E1 -19777.998,E2 -19777.998} C_VEL
LIN {X 0,Y 267.786,Z 197.008,A -85,B 0,C 180,E1 -19780.415,E2 -19780.415} C_VEL
LIN {X 0,Y 264.343,Z 192.423,A -85,B 0,C 180,E1 -19781.921,E2 -19781.921} C_VEL
LIN {X 0,Y 261.642,Z 188.731,A -85,B 0,C 180,E1 -19783.204,E2 -19783.204} C_VEL
LIN {X 0,Y 258.21,Z 184.215,A -85,B 0,C 180,E1 -19784.963,E2 -19784.963} C_VEL
LIN {X 0,Y 255.433,Z 180.753,A -85,B 0,C 180,E1 -19786.5,E2 -19786.5} C_VEL
LIN {X 0,Y 254.7,Z 179.607,A -85,B 0,C 180,E1 -19786.942,E2 -19786.942} C_VEL
LIN {X 0,Y 251.875,Z 176.763,A -85,B 0,C 180,E1 -19788.634,E2 -19788.634} C_VEL
LIN {X 0,Y 250.294,Z 174.216,A -85,B 0,C 180,E1 -19789.739,E2 -19789.739} C_VEL
LIN {X 0,Y 247.756,Z 171.833,A -85,B 0,C 180,E1 -19791.55,E2 -19791.55} C_VEL
LIN {X 0,Y 246.066,Z 168.723,A -85,B 0,C 180,E1 -19793.027,E2 -19793.027} C_VEL
LIN {X 0,Y 243.834,Z 167.609,A -85,B 0,C 180,E1 -19794.905,E2 -19794.905} C_VEL
LIN {X 0,Y 242.405,Z 167.017,A -85,B 0,C 180,E1 -19796.259,E2 -19796.259} C_VEL
LIN {X 0,Y 240.14,Z 167.589,A -85,B 0,C 180,E1 -19798.557,E2 -19798.557} C_VEL
LIN {X 0,Y 237.905,Z 168.673,A -85,B 0,C 180,E1 -19801.379,E2 -19801.379} C_VEL
LIN {X 0,Y 237.357,Z 168.632,A -85,B 0,C 180,E1 -19802.335,E2 -19802.335} C_VEL
LIN {X 0,Y 235.684,Z 167.042,A -85,B 0,C 180,E1 -19808.574,E2 -19808.574} C_VEL
LIN {X 0,Y 236.758,Z 168.461,A -85,B 0,C 180,E1 -19815.054,E2 -19815.054} C_VEL
LIN {X 0,Y 239.568,Z 170.207,A -85,B 0,C 180,E1 -19819.828,E2 -19819.828} C_VEL
LIN {X 0,Y 240.828,Z 172.924,A -85,B 0,C 180,E1 -19821.616,E2 -19821.616} C_VEL
LIN {X 0,Y 243.431,Z 175.547,A -85,B 0,C 180,E1 -19824.291,E2 -19824.291} C_VEL
LIN {X 0,Y 246.093,Z 178.823,A -85,B 0,C 180,E1 -19826.615,E2 -19826.615} C_VEL
LIN {X 0,Y 248.778,Z 182.683,A -85,B 0,C 180,E1 -19828.701,E2 -19828.701} C_VEL
LIN {X 0,Y 250.048,Z 184.238,A -85,B 0,C 180,E1 -19829.574,E2 -19829.574} C_VEL
LIN {X 0,Y 254.959,Z 191.21,A -85,B 0,C 180,E1 -19832.639,E2 -19832.639} C_VEL
LIN {X 0,Y 258.907,Z 197.269,A -85,B 0,C 180,E1 -19834.82,E2 -19834.82} C_VEL
LIN {X 0,Y 262.685,Z 203.121,A -85,B 0,C 180,E1 -19836.701,E2 -19836.701} C_VEL
LIN {X 0,Y 269.1,Z 213.968,A -85,B 0,C 180,E1 -19839.557,E2 -19839.557} C_VEL
LIN {X 0,Y 274.219,Z 223.527,A -85,B 0,C 180,E1 -19841.635,E2 -19841.635} C_VEL
LIN {X 0,Y 279.108,Z 233.647,A -85,B 0,C 180,E1 -19843.5,E2 -19843.5} C_VEL
LIN {X 0,Y 281.982,Z 240.219,A -85,B 0,C 180,E1 -19844.537,E2 -19844.537} C_VEL
LIN {X 0,Y 276.306,Z 325.965,A -85,B 0,C 180,E1 -19846.689,E2 -19846.689} C_VEL
LIN {X 0,Y 274.25,Z 341.726,A -85,B 0,C 180,E1 -19847.29,E2 -19847.29} C_VEL
LIN {X 0,Y 271.487,Z 356.201,A -85,B 0,C 180,E1 -19848.072,E2 -19848.072} C_VEL
LIN {X 0,Y 268.224,Z 369.882,A -85,B 0,C 180,E1 -19849.077,E2 -19849.077} C_VEL
LIN {X 0,Y 264.39,Z 383.349,A -85,B 0,C 180,E1 -19850.36,E2 -19850.36} C_VEL
LIN {X 0,Y 260.243,Z 395.793,A -85,B 0,C 180,E1 -19851.849,E2 -19851.849} C_VEL
LIN {X 0,Y 255.551,Z 408.438,A -85,B 0,C 180,E1 -19853.753,E2 -19853.753} C_VEL
LIN {X 0,Y 250.64,Z 419.973,A -85,B 0,C 180,E1 -19855.889,E2 -19855.889} C_VEL
LIN {X 0,Y 245.491,Z 431.19,A -85,B 0,C 180,E1 -19858.503,E2 -19858.503} C_VEL
LIN {X 0,Y 240.793,Z 440.689,A -85,B 0,C 180,E1 -19861.272,E2 -19861.272} C_VEL
LIN {X 0,Y 237.003,Z 448.352,A -85,B 0,C 180,E1 -19864.063,E2 -19864.063} C_VEL
LIN {X 0,Y 233.635,Z 454.898,A -85,B 0,C 180,E1 -19866.981,E2 -19866.981} C_VEL
LIN {X 0,Y 230.486,Z 460.949,A -85,B 0,C 180,E1 -19870.403,E2 -19870.403} C_VEL
LIN {X 0,Y 228.203,Z 465.643,A -85,B 0,C 180,E1 -19873.909,E2 -19873.909} C_VEL
LIN {X 0,Y 226.675,Z 469.107,A -85,B 0,C 180,E1 -19877.466,E2 -19877.466} C_VEL
LIN {X 0,Y 225.874,Z 471.412,A -85,B 0,C 180,E1 -19881.051,E2 -19881.051} C_VEL
LIN {X 0,Y 225.56,Z 472.599,A -85,B 0,C 180,E1 -19884.637,E2 -19884.637} C_VEL
LIN {X 0,Y 225.65,Z 472.648,A -85,B 0,C 180,E1 -19888.216,E2 -19888.216} C_VEL
LIN {X 0,Y 225.732,Z 472.219,A -85,B 0,C 180,E1 -19890.001,E2 -19890.001} C_VEL
LIN {X 0,Y 225.606,Z 470.475,A -85,B 0,C 180,E1 -19893.573,E2 -19893.573} C_VEL
LIN {X 0,Y 225.7,Z 467.522,A -85,B 0,C 180,E1 -19897.156,E2 -19897.156} C_VEL
LIN {X 0,Y 226.1,Z 463.272,A -85,B 0,C 180,E1 -19900.749,E2 -19900.749} C_VEL
LIN {X 0,Y 227.103,Z 457.615,A -85,B 0,C 180,E1 -19904.335,E2 -19904.335} C_VEL
LIN {X 0,Y 228.685,Z 450.386,A -85,B 0,C 180,E1 -19907.899,E2 -19907.899} C_VEL
LIN {X 0,Y 230.658,Z 442.624,A -85,B 0,C 180,E1 -19910.979,E2 -19910.979} C_VEL
LIN {X 0,Y 233.313,Z 433.264,A -85,B 0,C 180,E1 -19913.996,E2 -19913.996} C_VEL
LIN {X 0,Y 236.071,Z 422.912,A -85,B 0,C 180,E1 -19916.733,E2 -19916.733} C_VEL
LIN {X 0,Y 239.272,Z 411.263,A -85,B 0,C 180,E1 -19919.231,E2 -19919.231} C_VEL
LIN {X 0,Y 242.425,Z 398.52,A -85,B 0,C 180,E1 -19921.456,E2 -19921.456} C_VEL
LIN {X 0,Y 245.43,Z 386.016,A -85,B 0,C 180,E1 -19923.207,E2 -19923.207} C_VEL
LIN {X 0,Y 248.164,Z 372.994,A -85,B 0,C 180,E1 -19924.672,E2 -19924.672} C_VEL
LIN {X 0,Y 250.586,Z 358.593,A -85,B 0,C 180,E1 -19925.96,E2 -19925.96} C_VEL
LIN {X 0,Y 252.814,Z 343.314,A -85,B 0,C 180,E1 -19926.954,E2 -19926.954} C_VEL
LIN {X 0,Y 254.377,Z 327.163,A -85,B 0,C 180,E1 -19927.683,E2 -19927.683} C_VEL
LIN {X 0,Y 259.311,Z 225.148,A -85,B 0,C 180,E1 -19930.448,E2 -19930.448} C_VEL
LIN {X 0,Y 256.883,Z 218.233,A -85,B 0,C 180,E1 -19931.055,E2 -19931.055} C_VEL
LIN {X 0,Y 248.732,Z 198.679,A -85,B 0,C 180,E1 -19933.059,E2 -19933.059} C_VEL
LIN {X 0,Y 241.726,Z 184,A -85,B 0,C 180,E1 -19934.856,E2 -19934.856} C_VEL
LIN {X 0,Y 233.496,Z 168.751,A -85,B 0,C 180,E1 -19937.08,E2 -19937.08} C_VEL
LIN {X 0,Y 230.482,Z 163.618,A -85,B 0,C 180,E1 -19937.932,E2 -19937.932} C_VEL
LIN {X 0,Y 228.456,Z 159.839,A -85,B 0,C 180,E1 -19938.594,E2 -19938.594} C_VEL
LIN {X 0,Y 227.827,Z 157.725,A -85,B 0,C 180,E1 -19939.624,E2 -19939.624} C_VEL
LIN {X 0,Y 227.883,Z 157.72,A -85,B 0,C 180,E1 -19944.129,E2 -19944.129} C_VEL
LIN {X 0,Y 227.858,Z 157.726,A -85,B 0,C 180,E1 -19948.377,E2 -19948.377} C_VEL
LIN {X 0,Y 227.857,Z 157.691,A -85,B 0,C 180,E1 -19952.442,E2 -19952.442} C_VEL
LIN {X 0,Y 227.897,Z 157.721,A -85,B 0,C 180,E1 -19956.366,E2 -19956.366} C_VEL
LIN {X 0,Y 227.928,Z 157.716,A -85,B 0,C 180,E1 -19960.174,E2 -19960.174} C_VEL
LIN {X 0,Y 228.033,Z 157.697,A -85,B 0,C 180,E1 -19963.897,E2 -19963.897} C_VEL
LIN {X 0,Y 228.062,Z 157.692,A -85,B 0,C 180,E1 -19967.543,E2 -19967.543} C_VEL
LIN {X 0,Y 228.257,Z 157.673,A -85,B 0,C 180,E1 -19971.145,E2 -19971.145} C_VEL
LIN {X 0,Y 228.305,Z 157.663,A -85,B 0,C 180,E1 -19972.928,E2 -19972.928} C_VEL
LIN {X 0,Y 228.539,Z 157.604,A -85,B 0,C 180,E1 -19978.238,E2 -19978.238} C_VEL
LIN {X 0,Y 228.536,Z 157.617,A -85,B 0,C 180,E1 -19981.763,E2 -19981.763} C_VEL
LIN {X 0,Y 228.303,Z 157.647,A -85,B 0,C 180,E1 -19987.074,E2 -19987.074} C_VEL
LIN {X 0,Y 228.128,Z 157.651,A -85,B 0,C 180,E1 -19990.653,E2 -19990.653} C_VEL
LIN {X 0,Y 228.003,Z 157.7,A -85,B 0,C 180,E1 -19996.107,E2 -19996.107} C_VEL
LIN {X 0,Y 227.921,Z 157.709,A -85,B 0,C 180,E1 -20001.718,E2 -20001.718} C_VEL
LIN {X 0,Y 227.905,Z 157.707,A -85,B 0,C 180,E1 -20006.581,E2 -20006.581} C_VEL
LIN {X 0,Y 227.874,Z 157.685,A -85,B 0,C 180,E1 -20010.279,E2 -20010.279} C_VEL
LIN {X 0,Y 227.881,Z 157.723,A -85,B 0,C 180,E1 -20013.721,E2 -20013.721} C_VEL
LIN {X 0,Y 227.845,Z 157.691,A -85,B 0,C 180,E1 -20018.092,E2 -20018.092} C_VEL
LIN {X 0,Y 227.797,Z 157.733,A -85,B 0,C 180,E1 -20022.747,E2 -20022.747} C_VEL
LIN {X 0,Y 227.788,Z 157.715,A -85,B 0,C 180,E1 -20027.251,E2 -20027.251} C_VEL
LIN {X 0,Y 227.842,Z 157.708,A -85,B 0,C 180,E1 -20031.907,E2 -20031.907} C_VEL
LIN {X 0,Y 227.883,Z 157.713,A -85,B 0,C 180,E1 -20036.378,E2 -20036.378} C_VEL
LIN {X 0,Y 227.88,Z 157.72,A -85,B 0,C 180,E1 -20040.686,E2 -20040.686} C_VEL
LIN {X 0,Y 228.868,Z 160.548,A -85,B 0,C 180,E1 -20041.057,E2 -20041.057} C_VEL
LIN {X 0,Y 230.845,Z 163.072,A -85,B 0,C 180,E1 -20041.596,E2 -20041.596} C_VEL
LIN {X 0,Y 239.103,Z 176.119,A -85,B 0,C 180,E1 -20043.815,E2 -20043.815} C_VEL
LIN {X 0,Y 248.18,Z 191.538,A -85,B 0,C 180,E1 -20046.063,E2 -20046.063} C_VEL
LIN {X 0,Y 253.164,Z 201.286,A -85,B 0,C 180,E1 -20047.247,E2 -20047.247} C_VEL
LIN {X 0,Y 259.504,Z 216.569,A -85,B 0,C 180,E1 -20048.762,E2 -20048.762} C_VEL
LIN {X 0,Y 254.655,Z 315.491,A -85,B 0,C 180,E1 -20051.443,E2 -20051.443} C_VEL
LIN {X 0,Y 253.195,Z 331.254,A -85,B 0,C 180,E1 -20052.169,E2 -20052.169} C_VEL
LIN {X 0,Y 251.402,Z 345.719,A -85,B 0,C 180,E1 -20053.139,E2 -20053.139} C_VEL
LIN {X 0,Y 248.965,Z 360.422,A -85,B 0,C 180,E1 -20054.444,E2 -20054.444} C_VEL
LIN {X 0,Y 246.403,Z 373.775,A -85,B 0,C 180,E1 -20055.972,E2 -20055.972} C_VEL
LIN {X 0,Y 243.292,Z 387.389,A -85,B 0,C 180,E1 -20057.91,E2 -20057.91} C_VEL
LIN {X 0,Y 240.123,Z 399.76,A -85,B 0,C 180,E1 -20060.098,E2 -20060.098} C_VEL
LIN {X 0,Y 236.879,Z 411.843,A -85,B 0,C 180,E1 -20062.755,E2 -20062.755} C_VEL
LIN {X 0,Y 234.223,Z 421.239,A -85,B 0,C 180,E1 -20065.266,E2 -20065.266} C_VEL
LIN {X 0,Y 231.692,Z 430.423,A -85,B 0,C 180,E1 -20068.261,E2 -20068.261} C_VEL
LIN {X 0,Y 229.559,Z 438.072,A -85,B 0,C 180,E1 -20071.315,E2 -20071.315} C_VEL
LIN {X 0,Y 227.983,Z 444.395,A -85,B 0,C 180,E1 -20074.419,E2 -20074.419} C_VEL
LIN {X 0,Y 226.681,Z 450.138,A -85,B 0,C 180,E1 -20077.968,E2 -20077.968} C_VEL
LIN {X 0,Y 226.006,Z 453.689,A -85,B 0,C 180,E1 -20080.753,E2 -20080.753} C_VEL
LIN {X 0,Y 225.471,Z 457.12,A -85,B 0,C 180,E1 -20084.439,E2 -20084.439} C_VEL
LIN {X 0,Y 225.239,Z 459.301,A -85,B 0,C 180,E1 -20088.181,E2 -20088.181} C_VEL
LIN {X 0,Y 225.315,Z 460.085,A -85,B 0,C 180,E1 -20090.647,E2 -20090.647} C_VEL
LIN {X 0,Y 225.574,Z 460.232,A -85,B 0,C 180,E1 -20093.892,E2 -20093.892} C_VEL
LIN {X 0,Y 226.318,Z 459.251,A -85,B 0,C 180,E1 -20097.762,E2 -20097.762} C_VEL
LIN {X 0,Y 227.736,Z 456.922,A -85,B 0,C 180,E1 -20101.642,E2 -20101.642} C_VEL
LIN {X 0,Y 229.846,Z 453.158,A -85,B 0,C 180,E1 -20105.518,E2 -20105.518} C_VEL
LIN {X 0,Y 232.834,Z 447.859,A -85,B 0,C 180,E1 -20109.336,E2 -20109.336} C_VEL
LIN {X 0,Y 235.795,Z 442.542,A -85,B 0,C 180,E1 -20112.273,E2 -20112.273} C_VEL
LIN {X 0,Y 239.394,Z 435.898,A -85,B 0,C 180,E1 -20115.203,E2 -20115.203} C_VEL
LIN {X 0,Y 243.466,Z 427.944,A -85,B 0,C 180,E1 -20118.013,E2 -20118.013} C_VEL
LIN {X 0,Y 247.912,Z 418.935,A -85,B 0,C 180,E1 -20120.578,E2 -20120.578} C_VEL
LIN {X 0,Y 251.914,Z 410.101,A -85,B 0,C 180,E1 -20122.663,E2 -20122.663} C_VEL
LIN {X 0,Y 256.777,Z 398.4,A -85,B 0,C 180,E1 -20124.916,E2 -20124.916} C_VEL
LIN {X 0,Y 261.339,Z 386.242,A -85,B 0,C 180,E1 -20126.787,E2 -20126.787} C_VEL
LIN {X 0,Y 265.324,Z 374.049,A -85,B 0,C 180,E1 -20128.313,E2 -20128.313} C_VEL
LIN {X 0,Y 268.883,Z 361.272,A -85,B 0,C 180,E1 -20129.603,E2 -20129.603} C_VEL
LIN {X 0,Y 272.264,Z 346.532,A -85,B 0,C 180,E1 -20130.754,E2 -20130.754} C_VEL
LIN {X 0,Y 274.655,Z 333.064,A -85,B 0,C 180,E1 -20131.546,E2 -20131.546} C_VEL
LIN {X 0,Y 276.646,Z 317.86,A -85,B 0,C 180,E1 -20132.175,E2 -20132.175} C_VEL
LIN {X 0,Y 278.518,Z 291.231,A -85,B 0,C 180,E1 -20132.892,E2 -20132.892} C_VEL
LIN {X 0,Y 282.349,Z 232.958,A -85,B 0,C 180,E1 -20134.327,E2 -20134.327} C_VEL
LIN {X 0,Y 276.529,Z 221.346,A -85,B 0,C 180,E1 -20136.441,E2 -20136.441} C_VEL
LIN {X 0,Y 270.672,Z 210.962,A -85,B 0,C 180,E1 -20138.736,E2 -20138.736} C_VEL
LIN {X 0,Y 264.59,Z 202.122,A -85,B 0,C 180,E1 -20141.296,E2 -20141.296} C_VEL
LIN {X 0,Y 259.337,Z 194.865,A -85,B 0,C 180,E1 -20143.804,E2 -20143.804} C_VEL
LIN {X 0,Y 255.975,Z 190.422,A -85,B 0,C 180,E1 -20145.592,E2 -20145.592} C_VEL
LIN {X 0,Y 253.142,Z 186.599,A -85,B 0,C 180,E1 -20147.243,E2 -20147.243} C_VEL
LIN {X 0,Y 249.645,Z 182.585,A -85,B 0,C 180,E1 -20149.446,E2 -20149.446} C_VEL
LIN {X 0,Y 248.584,Z 180.844,A -85,B 0,C 180,E1 -20150.233,E2 -20150.233} C_VEL
LIN {X 0,Y 246.08,Z 178.322,A -85,B 0,C 180,E1 -20152.099,E2 -20152.099} C_VEL
LIN {X 0,Y 244.464,Z 175.52,A -85,B 0,C 180,E1 -20153.551,E2 -20153.551} C_VEL
LIN {X 0,Y 241.707,Z 173.686,A -85,B 0,C 180,E1 -20156.092,E2 -20156.092} C_VEL
LIN {X 0,Y 240.178,Z 171,A -85,B 0,C 180,E1 -20158.008,E2 -20158.008} C_VEL
LIN {X 0,Y 239.709,Z 169.717,A -85,B 0,C 180,E1 -20158.739,E2 -20158.739} C_VEL
LIN {X 0,Y 237.357,Z 168.632,A -85,B 0,C 180,E1 -20162.335,E2 -20162.335} C_VEL
LIN {X 0,Y 236.641,Z 168.917,A -85,B 0,C 180,E1 -20163.753,E2 -20163.753} C_VEL
LIN {X 0,Y 235.573,Z 171.099,A -85,B 0,C 180,E1 -20166.086,E2 -20166.086} C_VEL
LIN {X 0,Y 234.804,Z 173.872,A -85,B 0,C 180,E1 -20168.914,E2 -20168.914} C_VEL
LIN {X 0,Y 234.765,Z 174.23,A -85,B 0,C 180,E1 -20169.879,E2 -20169.879} C_VEL
LIN {X 0,Y 238.298,Z 176.902,A -85,B 0,C 180,E1 -20179.332,E2 -20179.332} C_VEL
LIN {X 0,Y 239.68,Z 179.85,A -85,B 0,C 180,E1 -20181.362,E2 -20181.362} C_VEL
LIN {X 0,Y 242.149,Z 182.426,A -85,B 0,C 180,E1 -20183.974,E2 -20183.974} C_VEL
LIN {X 0,Y 244.499,Z 185.407,A -85,B 0,C 180,E1 -20186.113,E2 -20186.113} C_VEL
LIN {X 0,Y 247.159,Z 189.318,A -85,B 0,C 180,E1 -20188.255,E2 -20188.255} C_VEL
LIN {X 0,Y 248.594,Z 191.341,A -85,B 0,C 180,E1 -20189.293,E2 -20189.293} C_VEL
LIN {X 0,Y 252.823,Z 197.405,A -85,B 0,C 180,E1 -20192.014,E2 -20192.014} C_VEL
LIN {X 0,Y 256.795,Z 203.698,A -85,B 0,C 180,E1 -20194.298,E2 -20194.298} C_VEL
LIN {X 0,Y 260.224,Z 209.183,A -85,B 0,C 180,E1 -20196.081,E2 -20196.081} C_VEL
LIN {X 0,Y 265.834,Z 218.907,A -85,B 0,C 180,E1 -20198.697,E2 -20198.697} C_VEL
LIN {X 0,Y 271.09,Z 228.956,A -85,B 0,C 180,E1 -20200.929,E2 -20200.929} C_VEL
LIN {X 0,Y 275.723,Z 238.857,A -85,B 0,C 180,E1 -20202.777,E2 -20202.777} C_VEL
LIN {X 0,Y 277.471,Z 242.994,A -85,B 0,C 180,E1 -20203.456,E2 -20203.456} C_VEL
LIN {X 0,Y 271.72,Z 326.168,A -85,B 0,C 180,E1 -20205.559,E2 -20205.559} C_VEL
LIN {X 0,Y 269.552,Z 341.984,A -85,B 0,C 180,E1 -20206.167,E2 -20206.167} C_VEL
LIN {X 0,Y 266.594,Z 356.944,A -85,B 0,C 180,E1 -20206.991,E2 -20206.991} C_VEL
LIN {X 0,Y 262.975,Z 371.395,A -85,B 0,C 180,E1 -20208.078,E2 -20208.078} C_VEL
LIN {X 0,Y 258.588,Z 385.889,A -85,B 0,C 180,E1 -20209.522,E2 -20209.522} C_VEL
LIN {X 0,Y 254.345,Z 397.999,A -85,B 0,C 180,E1 -20211.052,E2 -20211.052} C_VEL
LIN {X 0,Y 249.465,Z 410.244,A -85,B 0,C 180,E1 -20212.974,E2 -20212.974} C_VEL
LIN {X 0,Y 244.816,Z 420.568,A -85,B 0,C 180,E1 -20214.961,E2 -20214.961} C_VEL
LIN {X 0,Y 240.204,Z 430.183,A -85,B 0,C 180,E1 -20217.23,E2 -20217.23} C_VEL
LIN {X 0,Y 234.946,Z 440.247,A -85,B 0,C 180,E1 -20220.167,E2 -20220.167} C_VEL
LIN {X 0,Y 230.638,Z 448.603,A -85,B 0,C 180,E1 -20223.292,E2 -20223.292} C_VEL
LIN {X 0,Y 227.072,Z 455.06,A -85,B 0,C 180,E1 -20226.275,E2 -20226.275} C_VEL
LIN {X 0,Y 223.758,Z 461.041,A -85,B 0,C 180,E1 -20229.788,E2 -20229.788} C_VEL
LIN {X 0,Y 221.331,Z 465.676,A -85,B 0,C 180,E1 -20233.395,E2 -20233.395} C_VEL
LIN {X 0,Y 219.692,Z 469.06,A -85,B 0,C 180,E1 -20237.061,E2 -20237.061} C_VEL
LIN {X 0,Y 218.811,Z 471.294,A -85,B 0,C 180,E1 -20240.759,E2 -20240.759} C_VEL
LIN {X 0,Y 218.477,Z 472.414,A -85,B 0,C 180,E1 -20244.463,E2 -20244.463} C_VEL
LIN {X 0,Y 218.544,Z 472.42,A -85,B 0,C 180,E1 -20248.158,E2 -20248.158} C_VEL
LIN {X 0,Y 218.646,Z 471.97,A -85,B 0,C 180,E1 -20250.001,E2 -20250.001} C_VEL
LIN {X 0,Y 218.509,Z 470.158,A -85,B 0,C 180,E1 -20253.689,E2 -20253.689} C_VEL
LIN {X 0,Y 218.619,Z 467.134,A -85,B 0,C 180,E1 -20257.389,E2 -20257.389} C_VEL
LIN {X 0,Y 219.079,Z 462.811,A -85,B 0,C 180,E1 -20261.098,E2 -20261.098} C_VEL
LIN {X 0,Y 220.126,Z 457.072,A -85,B 0,C 180,E1 -20264.799,E2 -20264.799} C_VEL
LIN {X 0,Y 221.853,Z 449.759,A -85,B 0,C 180,E1 -20268.47,E2 -20268.47} C_VEL
LIN {X 0,Y 223.945,Z 441.9,A -85,B 0,C 180,E1 -20271.639,E2 -20271.639} C_VEL
LIN {X 0,Y 226.742,Z 432.431,A -85,B 0,C 180,E1 -20274.737,E2 -20274.737} C_VEL
LIN {X 0,Y 229.427,Z 422.749,A -85,B 0,C 180,E1 -20277.355,E2 -20277.355} C_VEL
LIN {X 0,Y 232.701,Z 411.24,A -85,B 0,C 180,E1 -20279.89,E2 -20279.89} C_VEL
LIN {X 0,Y 235.973,Z 398.535,A -85,B 0,C 180,E1 -20282.167,E2 -20282.167} C_VEL
LIN {X 0,Y 239.079,Z 386.07,A -85,B 0,C 180,E1 -20283.955,E2 -20283.955} C_VEL
LIN {X 0,Y 242.208,Z 371.41,A -85,B 0,C 180,E1 -20285.624,E2 -20285.624} C_VEL
LIN {X 0,Y 244.807,Z 356.444,A -85,B 0,C 180,E1 -20286.935,E2 -20286.935} C_VEL
LIN {X 0,Y 246.882,Z 341.951,A -85,B 0,C 180,E1 -20287.867,E2 -20287.867} C_VEL
LIN {X 0,Y 248.397,Z 326.372,A -85,B 0,C 180,E1 -20288.561,E2 -20288.561} C_VEL
LIN {X 0,Y 253.386,Z 226.443,A -85,B 0,C 180,E1 -20291.312,E2 -20291.312} C_VEL
LIN {X 0,Y 245.457,Z 206.581,A -85,B 0,C 180,E1 -20293.331,E2 -20293.331} C_VEL
LIN {X 0,Y 237.982,Z 190.226,A -85,B 0,C 180,E1 -20295.323,E2 -20295.323} C_VEL
LIN {X 0,Y 229.248,Z 173.696,A -85,B 0,C 180,E1 -20297.779,E2 -20297.779} C_VEL
LIN {X 0,Y 226.061,Z 168.221,A -85,B 0,C 180,E1 -20298.72,E2 -20298.72} C_VEL
LIN {X 0,Y 223.137,Z 163.48,A -85,B 0,C 180,E1 -20299.596,E2 -20299.596} C_VEL
LIN {X 0,Y 221.136,Z 159.996,A -85,B 0,C 180,E1 -20300.226,E2 -20300.226} C_VEL
LIN {X 0,Y 220.806,Z 158.591,A -85,B 0,C 180,E1 -20300.833,E2 -20300.833} C_VEL
LIN {X 0,Y 220.803,Z 158.603,A -85,B 0,C 180,E1 -20305.046,E2 -20305.046} C_VEL
LIN {X 0,Y 220.836,Z 158.599,A -85,B 0,C 180,E1 -20309.391,E2 -20309.391} C_VEL
LIN {X 0,Y 220.878,Z 158.565,A -85,B 0,C 180,E1 -20313.548,E2 -20313.548} C_VEL
LIN {X 0,Y 220.87,Z 158.589,A -85,B 0,C 180,E1 -20317.553,E2 -20317.553} C_VEL
LIN {X 0,Y 220.966,Z 158.574,A -85,B 0,C 180,E1 -20322.591,E2 -20322.591} C_VEL
LIN {X 0,Y 221.001,Z 158.573,A -85,B 0,C 180,E1 -20327.139,E2 -20327.139} C_VEL
LIN {X 0,Y 221.198,Z 158.554,A -85,B 0,C 180,E1 -20330.86,E2 -20330.86} C_VEL
LIN {X 0,Y 221.242,Z 158.542,A -85,B 0,C 180,E1 -20332.701,E2 -20332.701} C_VEL
LIN {X 0,Y 221.472,Z 158.484,A -85,B 0,C 180,E1 -20338.182,E2 -20338.182} C_VEL
LIN {X 0,Y 221.469,Z 158.497,A -85,B 0,C 180,E1 -20341.819,E2 -20341.819} C_VEL
LIN {X 0,Y 221.24,Z 158.523,A -85,B 0,C 180,E1 -20347.301,E2 -20347.301} C_VEL
LIN {X 0,Y 221.053,Z 158.535,A -85,B 0,C 180,E1 -20350.998,E2 -20350.998} C_VEL
LIN {X 0,Y 220.97,Z 158.574,A -85,B 0,C 180,E1 -20356.634,E2 -20356.634} C_VEL
LIN {X 0,Y 220.847,Z 158.598,A -85,B 0,C 180,E1 -20360.491,E2 -20360.491} C_VEL
LIN {X 0,Y 220.807,Z 158.605,A -85,B 0,C 180,E1 -20364.443,E2 -20364.443} C_VEL
LIN {X 0,Y 220.8,Z 158.566,A -85,B 0,C 180,E1 -20368.52,E2 -20368.52} C_VEL
LIN {X 0,Y 220.816,Z 158.597,A -85,B 0,C 180,E1 -20372.757,E2 -20372.757} C_VEL
LIN {X 0,Y 220.806,Z 158.571,A -85,B 0,C 180,E1 -20377.275,E2 -20377.275} C_VEL
LIN {X 0,Y 220.759,Z 158.61,A -85,B 0,C 180,E1 -20381.956,E2 -20381.956} C_VEL
LIN {X 0,Y 220.758,Z 158.582,A -85,B 0,C 180,E1 -20385.541,E2 -20385.541} C_VEL
LIN {X 0,Y 220.785,Z 158.6,A -85,B 0,C 180,E1 -20390.457,E2 -20390.457} C_VEL
LIN {X 0,Y 220.83,Z 158.582,A -85,B 0,C 180,E1 -20392.793,E2 -20392.793} C_VEL
LIN {X 0,Y 220.817,Z 158.589,A -85,B 0,C 180,E1 -20397.243,E2 -20397.243} C_VEL
LIN {X 0,Y 220.834,Z 158.599,A -85,B 0,C 180,E1 -20399.097,E2 -20399.097} C_VEL
LIN {X 0,Y 221.816,Z 161.441,A -85,B 0,C 180,E1 -20399.477,E2 -20399.477} C_VEL
LIN {X 0,Y 223.816,Z 163.929,A -85,B 0,C 180,E1 -20400.057,E2 -20400.057} C_VEL
LIN {X 0,Y 226.166,Z 167.414,A -85,B 0,C 180,E1 -20400.745,E2 -20400.745} C_VEL
LIN {X 0,Y 234.225,Z 180.122,A -85,B 0,C 180,E1 -20403.004,E2 -20403.004} C_VEL
LIN {X 0,Y 243.493,Z 196.063,A -85,B 0,C 180,E1 -20405.405,E2 -20405.405} C_VEL
LIN {X 0,Y 248.095,Z 205.209,A -85,B 0,C 180,E1 -20406.547,E2 -20406.547} C_VEL
LIN {X 0,Y 253.647,Z 218.652,A -85,B 0,C 180,E1 -20407.932,E2 -20407.932} C_VEL
LIN {X 0,Y 248.624,Z 315.892,A -85,B 0,C 180,E1 -20410.6,E2 -20410.6} C_VEL
LIN {X 0,Y 247.119,Z 331.591,A -85,B 0,C 180,E1 -20411.339,E2 -20411.339} C_VEL
LIN {X 0,Y 245.169,Z 346.607,A -85,B 0,C 180,E1 -20412.374,E2 -20412.374} C_VEL
LIN {X 0,Y 242.834,Z 360.264,A -85,B 0,C 180,E1 -20413.609,E2 -20413.609} C_VEL
LIN {X 0,Y 240.076,Z 374.089,A -85,B 0,C 180,E1 -20415.216,E2 -20415.216} C_VEL
LIN {X 0,Y 236.935,Z 387.376,A -85,B 0,C 180,E1 -20417.145,E2 -20417.145} C_VEL
LIN {X 0,Y 233.673,Z 399.78,A -85,B 0,C 180,E1 -20419.384,E2 -20419.384} C_VEL
LIN {X 0,Y 230.274,Z 411.905,A -85,B 0,C 180,E1 -20422.105,E2 -20422.105} C_VEL
LIN {X 0,Y 227.51,Z 421.313,A -85,B 0,C 180,E1 -20424.682,E2 -20424.682} C_VEL
LIN {X 0,Y 224.818,Z 430.688,A -85,B 0,C 180,E1 -20427.821,E2 -20427.821} C_VEL
LIN {X 0,Y 222.639,Z 438.186,A -85,B 0,C 180,E1 -20430.904,E2 -20430.904} C_VEL
LIN {X 0,Y 220.785,Z 445.35,A -85,B 0,C 180,E1 -20434.564,E2 -20434.564} C_VEL
LIN {X 0,Y 219.506,Z 450.991,A -85,B 0,C 180,E1 -20438.282,E2 -20438.282} C_VEL
LIN {X 0,Y 218.832,Z 454.334,A -85,B 0,C 180,E1 -20441.109,E2 -20441.109} C_VEL
LIN {X 0,Y 218.303,Z 457.71,A -85,B 0,C 180,E1 -20445.021,E2 -20445.021} C_VEL
LIN {X 0,Y 218.152,Z 459.701,A -85,B 0,C 180,E1 -20448.793,E2 -20448.793} C_VEL
LIN {X 0,Y 218.238,Z 460.299,A -85,B 0,C 180,E1 -20450.947,E2 -20450.947} C_VEL
LIN {X 0,Y 218.611,Z 460.404,A -85,B 0,C 180,E1 -20454.703,E2 -20454.703} C_VEL
LIN {X 0,Y 219.489,Z 459.265,A -85,B 0,C 180,E1 -20458.704,E2 -20458.704} C_VEL
LIN {X 0,Y 221.109,Z 456.777,A -85,B 0,C 180,E1 -20462.707,E2 -20462.707} C_VEL
LIN {X 0,Y 223.509,Z 452.851,A -85,B 0,C 180,E1 -20466.686,E2 -20466.686} C_VEL
LIN {X 0,Y 226.777,Z 447.374,A -85,B 0,C 180,E1 -20470.602,E2 -20470.602} C_VEL
LIN {X 0,Y 229.857,Z 442.134,A -85,B 0,C 180,E1 -20473.467,E2 -20473.467} C_VEL
LIN {X 0,Y 234.097,Z 434.654,A -85,B 0,C 180,E1 -20476.72,E2 -20476.72} C_VEL
LIN {X 0,Y 238.624,Z 426.267,A -85,B 0,C 180,E1 -20479.612,E2 -20479.612} C_VEL
LIN {X 0,Y 242.918,Z 417.866,A -85,B 0,C 180,E1 -20481.962,E2 -20481.962} C_VEL
LIN {X 0,Y 248.132,Z 406.623,A -85,B 0,C 180,E1 -20484.518,E2 -20484.518} C_VEL
LIN {X 0,Y 253.274,Z 394.408,A -85,B 0,C 180,E1 -20486.712,E2 -20486.712} C_VEL
LIN {X 0,Y 258.105,Z 381.332,A -85,B 0,C 180,E1 -20488.579,E2 -20488.579} C_VEL
LIN {X 0,Y 262.351,Z 367.661,A -85,B 0,C 180,E1 -20490.143,E2 -20490.143} C_VEL
LIN {X 0,Y 265.887,Z 354.285,A -85,B 0,C 180,E1 -20491.332,E2 -20491.332} C_VEL
LIN {X 0,Y 269.082,Z 338.708,A -85,B 0,C 180,E1 -20492.398,E2 -20492.398} C_VEL
LIN {X 0,Y 271.47,Z 323.461,A -85,B 0,C 180,E1 -20493.118,E2 -20493.118} C_VEL
LIN {X 0,Y 272.966,Z 307.57,A -85,B 0,C 180,E1 -20493.625,E2 -20493.625} C_VEL
LIN {X 0,Y 277.869,Z 235.986,A -85,B 0,C 180,E1 -20495.402,E2 -20495.402} C_VEL
LIN {X 0,Y 272.985,Z 226.081,A -85,B 0,C 180,E1 -20497.283,E2 -20497.283} C_VEL
LIN {X 0,Y 267.749,Z 216.602,A -85,B 0,C 180,E1 -20499.426,E2 -20499.426} C_VEL
LIN {X 0,Y 262.5,Z 208.777,A -85,B 0,C 180,E1 -20501.714,E2 -20501.714} C_VEL
LIN {X 0,Y 257.282,Z 201.301,A -85,B 0,C 180,E1 -20504.299,E2 -20504.299} C_VEL
LIN {X 0,Y 253.861,Z 196.688,A -85,B 0,C 180,E1 -20506.185,E2 -20506.185} C_VEL
LIN {X 0,Y 250.65,Z 192.414,A -85,B 0,C 180,E1 -20508.134,E2 -20508.134} C_VEL
LIN {X 0,Y 247.798,Z 188.937,A -85,B 0,C 180,E1 -20510.04,E2 -20510.04} C_VEL
LIN {X 0,Y 246.823,Z 187.434,A -85,B 0,C 180,E1 -20510.782,E2 -20510.782} C_VEL
LIN {X 0,Y 244.136,Z 184.362,A -85,B 0,C 180,E1 -20512.913,E2 -20512.913} C_VEL
LIN {X 0,Y 243.02,Z 182.347,A -85,B 0,C 180,E1 -20513.982,E2 -20513.982} C_VEL
LIN {X 0,Y 240.359,Z 180.407,A -85,B 0,C 180,E1 -20516.542,E2 -20516.542} C_VEL
LIN {X 0,Y 238.796,Z 177.462,A -85,B 0,C 180,E1 -20518.629,E2 -20518.629} C_VEL
LIN {X 0,Y 238.466,Z 176.665,A -85,B 0,C 180,E1 -20519.155,E2 -20519.155} C_VEL
LIN {X 0,Y 234.787,Z 174.088,A -85,B 0,C 180,E1 -20528.607,E2 -20528.607} C_VEL
LIN {X 0,Y 234.765,Z 174.23,A -85,B 0,C 180,E1 -20529.879,E2 -20529.879} C_VEL
LIN {X 0,Y 234.8,Z 175.132,A -85,B 0,C 180,E1 -20531.303,E2 -20531.303} C_VEL
LIN {X 0,Y 234.906,Z 178.592,A -85,B 0,C 180,E1 -20533.572,E2 -20533.572} C_VEL
LIN {X 0,Y 235.374,Z 182.2,A -85,B 0,C 180,E1 -20535.833,E2 -20535.833} C_VEL
LIN {X 0,Y 235.997,Z 183.326,A -85,B 0,C 180,E1 -20537.241,E2 -20537.241} C_VEL
LIN {X 0,Y 237.198,Z 184.065,A -85,B 0,C 180,E1 -20539.11,E2 -20539.11} C_VEL
LIN {X 0,Y 238.64,Z 186.945,A -85,B 0,C 180,E1 -20541.241,E2 -20541.241} C_VEL
LIN {X 0,Y 240.872,Z 189.307,A -85,B 0,C 180,E1 -20543.652,E2 -20543.652} C_VEL
LIN {X 0,Y 242.931,Z 191.978,A -85,B 0,C 180,E1 -20545.602,E2 -20545.602} C_VEL
LIN {X 0,Y 245.539,Z 195.937,A -85,B 0,C 180,E1 -20547.791,E2 -20547.791} C_VEL
LIN {X 0,Y 246.848,Z 197.865,A -85,B 0,C 180,E1 -20548.783,E2 -20548.783} C_VEL
LIN {X 0,Y 250.818,Z 203.778,A -85,B 0,C 180,E1 -20551.443,E2 -20551.443} C_VEL
LIN {X 0,Y 254.608,Z 209.955,A -85,B 0,C 180,E1 -20553.708,E2 -20553.708} C_VEL
LIN {X 0,Y 258.011,Z 215.55,A -85,B 0,C 180,E1 -20555.548,E2 -20555.548} C_VEL
LIN {X 0,Y 263.811,Z 225.999,A -85,B 0,C 180,E1 -20558.354,E2 -20558.354} C_VEL
LIN {X 0,Y 269.706,Z 237.934,A -85,B 0,C 180,E1 -20560.924,E2 -20560.924} C_VEL
LIN {X 0,Y 273.115,Z 246.078,A -85,B 0,C 180,E1 -20562.346,E2 -20562.346} C_VEL
LIN {X 0,Y 267.276,Z 326.403,A -85,B 0,C 180,E1 -20564.385,E2 -20564.385} C_VEL
LIN {X 0,Y 265.121,Z 341.619,A -85,B 0,C 180,E1 -20564.973,E2 -20564.973} C_VEL
LIN {X 0,Y 262.088,Z 356.577,A -85,B 0,C 180,E1 -20565.798,E2 -20565.798} C_VEL
LIN {X 0,Y 258.337,Z 371.031,A -85,B 0,C 180,E1 -20566.881,E2 -20566.881} C_VEL
LIN {X 0,Y 254.256,Z 384.185,A -85,B 0,C 180,E1 -20568.176,E2 -20568.176} C_VEL
LIN {X 0,Y 249.802,Z 396.41,A -85,B 0,C 180,E1 -20569.678,E2 -20569.678} C_VEL
LIN {X 0,Y 244.786,Z 408.881,A -85,B 0,C 180,E1 -20571.621,E2 -20571.621} C_VEL
LIN {X 0,Y 239.907,Z 419.399,A -85,B 0,C 180,E1 -20573.615,E2 -20573.615} C_VEL
LIN {X 0,Y 234.281,Z 430.646,A -85,B 0,C 180,E1 -20576.292,E2 -20576.292} C_VEL
LIN {X 0,Y 229.23,Z 439.911,A -85,B 0,C 180,E1 -20579.057,E2 -20579.057} C_VEL
LIN {X 0,Y 224.312,Z 448.854,A -85,B 0,C 180,E1 -20582.476,E2 -20582.476} C_VEL
LIN {X 0,Y 220.557,Z 455.221,A -85,B 0,C 180,E1 -20585.529,E2 -20585.529} C_VEL
LIN {X 0,Y 217.064,Z 461.12,A -85,B 0,C 180,E1 -20589.137,E2 -20589.137} C_VEL
LIN {X 0,Y 214.486,Z 465.704,A -85,B 0,C 180,E1 -20592.849,E2 -20592.849} C_VEL
LIN {X 0,Y 212.721,Z 469.022,A -85,B 0,C 180,E1 -20596.629,E2 -20596.629} C_VEL
LIN {X 0,Y 211.769,Z 471.181,A -85,B 0,C 180,E1 -20600.449,E2 -20600.449} C_VEL
LIN {X 0,Y 211.378,Z 472.23,A -85,B 0,C 180,E1 -20604.276,E2 -20604.276} C_VEL
LIN {X 0,Y 211.442,Z 472.173,A -85,B 0,C 180,E1 -20608.096,E2 -20608.096} C_VEL
LIN {X 0,Y 211.561,Z 471.714,A -85,B 0,C 180,E1 -20610.001,E2 -20610.001} C_VEL
LIN {X 0,Y 211.434,Z 469.843,A -85,B 0,C 180,E1 -20613.813,E2 -20613.813} C_VEL
LIN {X 0,Y 211.558,Z 466.748,A -85,B 0,C 180,E1 -20617.637,E2 -20617.637} C_VEL
LIN {X 0,Y 212.047,Z 462.349,A -85,B 0,C 180,E1 -20621.471,E2 -20621.471} C_VEL
LIN {X 0,Y 213.172,Z 456.529,A -85,B 0,C 180,E1 -20625.293,E2 -20625.293} C_VEL
LIN {X 0,Y 215.043,Z 449.128,A -85,B 0,C 180,E1 -20629.077,E2 -20629.077} C_VEL
LIN {X 0,Y 217.261,Z 441.166,A -85,B 0,C 180,E1 -20632.34,E2 -20632.34} C_VEL
LIN {X 0,Y 220.206,Z 431.577,A -85,B 0,C 180,E1 -20635.523,E2 -20635.523} C_VEL
LIN {X 0,Y 223.072,Z 421.758,A -85,B 0,C 180,E1 -20638.203,E2 -20638.203} C_VEL
LIN {X 0,Y 226.444,Z 410.068,A -85,B 0,C 180,E1 -20640.805,E2 -20640.805} C_VEL
LIN {X 0,Y 229.564,Z 398.47,A -85,B 0,C 180,E1 -20642.917,E2 -20642.917} C_VEL
LIN {X 0,Y 232.772,Z 386.014,A -85,B 0,C 180,E1 -20644.743,E2 -20644.743} C_VEL
LIN {X 0,Y 235.904,Z 371.914,A -85,B 0,C 180,E1 -20646.392,E2 -20646.392} C_VEL
LIN {X 0,Y 238.641,Z 356.739,A -85,B 0,C 180,E1 -20647.763,E2 -20647.763} C_VEL
LIN {X 0,Y 240.823,Z 342.07,A -85,B 0,C 180,E1 -20648.728,E2 -20648.728} C_VEL
LIN {X 0,Y 242.395,Z 326.695,A -85,B 0,C 180,E1 -20649.432,E2 -20649.432} C_VEL
LIN {X 0,Y 247.516,Z 228.416,A -85,B 0,C 180,E1 -20652.185,E2 -20652.185} C_VEL
LIN {X 0,Y 239.999,Z 209.433,A -85,B 0,C 180,E1 -20654.198,E2 -20654.198} C_VEL
LIN {X 0,Y 232.947,Z 193.882,A -85,B 0,C 180,E1 -20656.173,E2 -20656.173} C_VEL
LIN {X 0,Y 224.573,Z 177.885,A -85,B 0,C 180,E1 -20658.64,E2 -20658.64} C_VEL
LIN {X 0,Y 219.369,Z 168.959,A -85,B 0,C 180,E1 -20660.25,E2 -20660.25} C_VEL
LIN {X 0,Y 216.31,Z 164.084,A -85,B 0,C 180,E1 -20661.237,E2 -20661.237} C_VEL
LIN {X 0,Y 214.38,Z 161.638,A -85,B 0,C 180,E1 -20661.853,E2 -20661.853} C_VEL
LIN {X 0,Y 213.773,Z 159.472,A -85,B 0,C 180,E1 -20662.16,E2 -20662.16} C_VEL
LIN {X 0,Y 213.758,Z 159.484,A -85,B 0,C 180,E1 -20666.019,E2 -20666.019} C_VEL
LIN {X 0,Y 213.752,Z 159.462,A -85,B 0,C 180,E1 -20670.45,E2 -20670.45} C_VEL
LIN {X 0,Y 213.784,Z 159.463,A -85,B 0,C 180,E1 -20674.7,E2 -20674.7} C_VEL
LIN {X 0,Y 213.803,Z 159.466,A -85,B 0,C 180,E1 -20678.803,E2 -20678.803} C_VEL
LIN {X 0,Y 213.925,Z 159.451,A -85,B 0,C 180,E1 -20682.803,E2 -20682.803} C_VEL
LIN {X 0,Y 213.941,Z 159.455,A -85,B 0,C 180,E1 -20686.707,E2 -20686.707} C_VEL
LIN {X 0,Y 214.138,Z 159.435,A -85,B 0,C 180,E1 -20690.556,E2 -20690.556} C_VEL
LIN {X 0,Y 214.079,Z 159.443,A -85,B 0,C 180,E1 -20694.349,E2 -20694.349} C_VEL
LIN {X 0,Y 214.409,Z 159.363,A -85,B 0,C 180,E1 -20698.122,E2 -20698.122} C_VEL
LIN {X 0,Y 214.516,Z 159.342,A -85,B 0,C 180,E1 -20700.001,E2 -20700.001} C_VEL
LIN {X 0,Y 214.406,Z 159.376,A -85,B 0,C 180,E1 -20701.879,E2 -20701.879} C_VEL
LIN {X 0,Y 214.181,Z 159.397,A -85,B 0,C 180,E1 -20707.543,E2 -20707.543} C_VEL
LIN {X 0,Y 213.985,Z 159.419,A -85,B 0,C 180,E1 -20711.366,E2 -20711.366} C_VEL
LIN {X 0,Y 213.869,Z 159.468,A -85,B 0,C 180,E1 -20715.242,E2 -20715.242} C_VEL
LIN {X 0,Y 213.791,Z 159.478,A -85,B 0,C 180,E1 -20719.193,E2 -20719.193} C_VEL
LIN {X 0,Y 213.789,Z 159.473,A -85,B 0,C 180,E1 -20723.235,E2 -20723.235} C_VEL
LIN {X 0,Y 213.79,Z 159.451,A -85,B 0,C 180,E1 -20727.427,E2 -20727.427} C_VEL
LIN {X 0,Y 213.763,Z 159.459,A -85,B 0,C 180,E1 -20731.739,E2 -20731.739} C_VEL
LIN {X 0,Y 213.746,Z 159.461,A -85,B 0,C 180,E1 -20736.289,E2 -20736.289} C_VEL
LIN {X 0,Y 213.706,Z 159.482,A -85,B 0,C 180,E1 -20741.128,E2 -20741.128} C_VEL
LIN {X 0,Y 213.706,Z 159.478,A -85,B 0,C 180,E1 -20743.68,E2 -20743.68} C_VEL
LIN {X 0,Y 213.706,Z 159.46,A -85,B 0,C 180,E1 -20746.346,E2 -20746.346} C_VEL
LIN {X 0,Y 213.706,Z 159.491,A -85,B 0,C 180,E1 -20749.148,E2 -20749.148} C_VEL
LIN {X 0,Y 213.746,Z 159.471,A -85,B 0,C 180,E1 -20753.711,E2 -20753.711} C_VEL
LIN {X 0,Y 213.788,Z 159.482,A -85,B 0,C 180,E1 -20757.36,E2 -20757.36} C_VEL
LIN {X 0,Y 214.655,Z 162.097,A -85,B 0,C 180,E1 -20757.714,E2 -20757.714} C_VEL
LIN {X 0,Y 216.9,Z 164.862,A -85,B 0,C 180,E1 -20758.422,E2 -20758.422} C_VEL
LIN {X 0,Y 219.074,Z 168.173,A -85,B 0,C 180,E1 -20759.116,E2 -20759.116} C_VEL
LIN {X 0,Y 227.56,Z 181.134,A -85,B 0,C 180,E1 -20761.638,E2 -20761.638} C_VEL
LIN {X 0,Y 236.995,Z 197.157,A -85,B 0,C 180,E1 -20764.236,E2 -20764.236} C_VEL
LIN {X 0,Y 243.019,Z 208.996,A -85,B 0,C 180,E1 -20765.804,E2 -20765.804} C_VEL
LIN {X 0,Y 247.733,Z 220.494,A -85,B 0,C 180,E1 -20767.039,E2 -20767.039} C_VEL
LIN {X 0,Y 242.63,Z 316.141,A -85,B 0,C 180,E1 -20769.714,E2 -20769.714} C_VEL
LIN {X 0,Y 241.084,Z 331.813,A -85,B 0,C 180,E1 -20770.467,E2 -20770.467} C_VEL
LIN {X 0,Y 239.148,Z 346.263,A -85,B 0,C 180,E1 -20771.472,E2 -20771.472} C_VEL
LIN {X 0,Y 236.744,Z 359.993,A -85,B 0,C 180,E1 -20772.73,E2 -20772.73} C_VEL
LIN {X 0,Y 234.002,Z 373.468,A -85,B 0,C 180,E1 -20774.317,E2 -20774.317} C_VEL
LIN {X 0,Y 230.949,Z 385.968,A -85,B 0,C 180,E1 -20776.134,E2 -20776.134} C_VEL
LIN {X 0,Y 227.512,Z 398.659,A -85,B 0,C 180,E1 -20778.416,E2 -20778.416} C_VEL
LIN {X 0,Y 224.209,Z 410.161,A -85,B 0,C 180,E1 -20780.982,E2 -20780.982} C_VEL
LIN {X 0,Y 221.274,Z 419.849,A -85,B 0,C 180,E1 -20783.617,E2 -20783.617} C_VEL
LIN {X 0,Y 218.464,Z 429.266,A -85,B 0,C 180,E1 -20786.744,E2 -20786.744} C_VEL
LIN {X 0,Y 216.052,Z 437.257,A -85,B 0,C 180,E1 -20789.999,E2 -20789.999} C_VEL
LIN {X 0,Y 214.003,Z 444.648,A -85,B 0,C 180,E1 -20793.765,E2 -20793.765} C_VEL
LIN {X 0,Y 212.568,Z 450.498,A -85,B 0,C 180,E1 -20797.599,E2 -20797.599} C_VEL
LIN {X 0,Y 211.643,Z 454.957,A -85,B 0,C 180,E1 -20801.492,E2 -20801.492} C_VEL
LIN {X 0,Y 211.175,Z 458.12,A -85,B 0,C 180,E1 -20805.44,E2 -20805.44} C_VEL
LIN {X 0,Y 211.063,Z 460.04,A -85,B 0,C 180,E1 -20809.449,E2 -20809.449} C_VEL
LIN {X 0,Y 211.173,Z 460.534,A -85,B 0,C 180,E1 -20811.474,E2 -20811.474} C_VEL
LIN {X 0,Y 211.653,Z 460.569,A -85,B 0,C 180,E1 -20815.573,E2 -20815.573} C_VEL
LIN {X 0,Y 212.717,Z 459.286,A -85,B 0,C 180,E1 -20819.708,E2 -20819.708} C_VEL
LIN {X 0,Y 214.54,Z 456.637,A -85,B 0,C 180,E1 -20823.84,E2 -20823.84} C_VEL
LIN {X 0,Y 217.248,Z 452.544,A -85,B 0,C 180,E1 -20827.926,E2 -20827.926} C_VEL
LIN {X 0,Y 220.872,Z 446.889,A -85,B 0,C 180,E1 -20831.928,E2 -20831.928} C_VEL
LIN {X 0,Y 224.815,Z 440.484,A -85,B 0,C 180,E1 -20835.331,E2 -20835.331} C_VEL
LIN {X 0,Y 229.453,Z 432.557,A -85,B 0,C 180,E1 -20838.626,E2 -20838.626} C_VEL
LIN {X 0,Y 234.874,Z 422.873,A -85,B 0,C 180,E1 -20841.763,E2 -20841.763} C_VEL
LIN {X 0,Y 240.402,Z 411.973,A -85,B 0,C 180,E1 -20844.541,E2 -20844.541} C_VEL
LIN {X 0,Y 245.724,Z 400.356,A -85,B 0,C 180,E1 -20846.885,E2 -20846.885} C_VEL
LIN {X 0,Y 250.598,Z 388.491,A -85,B 0,C 180,E1 -20848.8,E2 -20848.8} C_VEL
LIN {X 0,Y 255.348,Z 375.107,A -85,B 0,C 180,E1 -20850.529,E2 -20850.529} C_VEL
LIN {X 0,Y 259.395,Z 361.608,A -85,B 0,C 180,E1 -20851.913,E2 -20851.913} C_VEL
LIN {X 0,Y 262.892,Z 347.445,A -85,B 0,C 180,E1 -20853.031,E2 -20853.031} C_VEL
LIN {X 0,Y 265.553,Z 333.654,A -85,B 0,C 180,E1 -20853.849,E2 -20853.849} C_VEL
LIN {X 0,Y 267.663,Z 318.752,A -85,B 0,C 180,E1 -20854.472,E2 -20854.472} C_VEL
LIN {X 0,Y 269.527,Z 294.794,A -85,B 0,C 180,E1 -20855.136,E2 -20855.136} C_VEL
LIN {X 0,Y 273.476,Z 238.965,A -85,B 0,C 180,E1 -20856.534,E2 -20856.534} C_VEL
LIN {X 0,Y 268.728,Z 229.244,A -85,B 0,C 180,E1 -20858.471,E2 -20858.471} C_VEL
LIN {X 0,Y 264.452,Z 221.553,A -85,B 0,C 180,E1 -20860.312,E2 -20860.312} C_VEL
LIN {X 0,Y 259.452,Z 213.936,A -85,B 0,C 180,E1 -20862.616,E2 -20862.616} C_VEL
LIN {X 0,Y 254.606,Z 206.935,A -85,B 0,C 180,E1 -20865.151,E2 -20865.151} C_VEL
LIN {X 0,Y 251.773,Z 202.97,A -85,B 0,C 180,E1 -20866.788,E2 -20866.788} C_VEL
LIN {X 0,Y 248.677,Z 198.775,A -85,B 0,C 180,E1 -20868.742,E2 -20868.742} C_VEL
LIN {X 0,Y 245.848,Z 195.067,A -85,B 0,C 180,E1 -20870.745,E2 -20870.745} C_VEL
LIN {X 0,Y 244.955,Z 193.874,A -85,B 0,C 180,E1 -20871.44,E2 -20871.44} C_VEL
LIN {X 0,Y 242.278,Z 190.4,A -85,B 0,C 180,E1 -20873.728,E2 -20873.728} C_VEL
LIN {X 0,Y 241.59,Z 189.172,A -85,B 0,C 180,E1 -20874.417,E2 -20874.417} C_VEL
LIN {X 0,Y 238.94,Z 186.999,A -85,B 0,C 180,E1 -20877.102,E2 -20877.102} C_VEL
LIN {X 0,Y 237.444,Z 183.925,A -85,B 0,C 180,E1 -20879.257,E2 -20879.257} C_VEL
LIN {X 0,Y 235.89,Z 182.874,A -85,B 0,C 180,E1 -20881.707,E2 -20881.707} C_VEL
LIN {X 0,Y 233.89,Z 181.135,A -85,B 0,C 180,E1 -20888.64,E2 -20888.64} C_VEL
LIN {X 0,Y 234.686,Z 182.357,A -85,B 0,C 180,E1 -20894.303,E2 -20894.303} C_VEL
LIN {X 0,Y 235.997,Z 183.326,A -85,B 0,C 180,E1 -20897.241,E2 -20897.241} C_VEL
LIN {X 0,Y 236.437,Z 184.484,A -85,B 0,C 180,E1 -20898.146,E2 -20898.146} C_VEL
LIN {X 0,Y 236.726,Z 186.754,A -85,B 0,C 180,E1 -20898.948,E2 -20898.948} C_VEL
LIN {X 0,Y 237.389,Z 192.899,A -85,B 0,C 180,E1 -20900.719,E2 -20900.719} C_VEL
LIN {X 0,Y 238.007,Z 194.5,A -85,B 0,C 180,E1 -20901.599,E2 -20901.599} C_VEL
LIN {X 0,Y 239.705,Z 196.297,A -85,B 0,C 180,E1 -20903.43,E2 -20903.43} C_VEL
LIN {X 0,Y 241.548,Z 198.869,A -85,B 0,C 180,E1 -20905.238,E2 -20905.238} C_VEL
LIN {X 0,Y 244.218,Z 202.873,A -85,B 0,C 180,E1 -20907.538,E2 -20907.538} C_VEL
LIN {X 0,Y 248.871,Z 210.176,A -85,B 0,C 180,E1 -20910.882,E2 -20910.882} C_VEL
LIN {X 0,Y 252.659,Z 216.56,A -85,B 0,C 180,E1 -20913.232,E2 -20913.232} C_VEL
LIN {X 0,Y 255.725,Z 221.795,A -85,B 0,C 180,E1 -20914.954,E2 -20914.954} C_VEL
LIN {X 0,Y 260.819,Z 231.297,A -85,B 0,C 180,E1 -20917.551,E2 -20917.551} C_VEL
LIN {X 0,Y 266.429,Z 242.98,A -85,B 0,C 180,E1 -20920.117,E2 -20920.117} C_VEL
LIN {X 0,Y 268.829,Z 248.668,A -85,B 0,C 180,E1 -20921.165,E2 -20921.165} C_VEL
LIN {X 0,Y 263.054,Z 326.137,A -85,B 0,C 180,E1 -20923.155,E2 -20923.155} C_VEL
LIN {X 0,Y 260.818,Z 341.411,A -85,B 0,C 180,E1 -20923.74,E2 -20923.74} C_VEL
LIN {X 0,Y 257.699,Z 356.37,A -85,B 0,C 180,E1 -20924.563,E2 -20924.563} C_VEL
LIN {X 0,Y 253.808,Z 370.833,A -85,B 0,C 180,E1 -20925.64,E2 -20925.64} C_VEL
LIN {X 0,Y 249.611,Z 383.965,A -85,B 0,C 180,E1 -20926.94,E2 -20926.94} C_VEL
LIN {X 0,Y 244.902,Z 396.361,A -85,B 0,C 180,E1 -20928.466,E2 -20928.466} C_VEL
LIN {X 0,Y 239.761,Z 408.606,A -85,B 0,C 180,E1 -20930.392,E2 -20930.392} C_VEL
LIN {X 0,Y 234.263,Z 419.993,A -85,B 0,C 180,E1 -20932.591,E2 -20932.591} C_VEL
LIN {X 0,Y 229.247,Z 429.636,A -85,B 0,C 180,E1 -20934.914,E2 -20934.914} C_VEL
LIN {X 0,Y 223.827,Z 439.143,A -85,B 0,C 180,E1 -20937.739,E2 -20937.739} C_VEL
LIN {X 0,Y 219.846,Z 446.07,A -85,B 0,C 180,E1 -20940.298,E2 -20940.298} C_VEL
LIN {X 0,Y 215.105,Z 453.744,A -85,B 0,C 180,E1 -20943.828,E2 -20943.828} C_VEL
LIN {X 0,Y 211.254,Z 459.887,A -85,B 0,C 180,E1 -20947.507,E2 -20947.507} C_VEL
LIN {X 0,Y 208.7,Z 463.841,A -85,B 0,C 180,E1 -20950.544,E2 -20950.544} C_VEL
LIN {X 0,Y 206.662,Z 467.504,A -85,B 0,C 180,E1 -20954.214,E2 -20954.214} C_VEL
LIN {X 0,Y 205.17,Z 470.168,A -85,B 0,C 180,E1 -20958.14,E2 -20958.14} C_VEL
LIN {X 0,Y 204.436,Z 471.696,A -85,B 0,C 180,E1 -20962.097,E2 -20962.097} C_VEL
LIN {X 0,Y 204.261,Z 472.114,A -85,B 0,C 180,E1 -20966.189,E2 -20966.189} C_VEL
LIN {X 0,Y 204.478,Z 471.43,A -85,B 0,C 180,E1 -20970.001,E2 -20970.001} C_VEL
LIN {X 0,Y 204.382,Z 469.299,A -85,B 0,C 180,E1 -20974.288,E2 -20974.288} C_VEL
LIN {X 0,Y 204.471,Z 466.347,A -85,B 0,C 180,E1 -20977.903,E2 -20977.903} C_VEL
LIN {X 0,Y 205.012,Z 461.866,A -85,B 0,C 180,E1 -20981.87,E2 -20981.87} C_VEL
LIN {X 0,Y 206.238,Z 455.957,A -85,B 0,C 180,E1 -20985.821,E2 -20985.821} C_VEL
LIN {X 0,Y 208.252,Z 448.461,A -85,B 0,C 180,E1 -20989.724,E2 -20989.724} C_VEL
LIN {X 0,Y 210.612,Z 440.395,A -85,B 0,C 180,E1 -20993.086,E2 -20993.086} C_VEL
LIN {X 0,Y 213.254,Z 432.207,A -85,B 0,C 180,E1 -20995.892,E2 -20995.892} C_VEL
LIN {X 0,Y 216.434,Z 421.74,A -85,B 0,C 180,E1 -20998.854,E2 -20998.854} C_VEL
LIN {X 0,Y 219.67,Z 411.061,A -85,B 0,C 180,E1 -21001.326,E2 -21001.326} C_VEL
LIN {X 0,Y 223.199,Z 398.388,A -85,B 0,C 180,E1 -21003.71,E2 -21003.71} C_VEL
LIN {X 0,Y 226.511,Z 385.948,A -85,B 0,C 180,E1 -21005.575,E2 -21005.575} C_VEL
LIN {X 0,Y 229.474,Z 373.153,A -85,B 0,C 180,E1 -21007.115,E2 -21007.115} C_VEL
LIN {X 0,Y 232.177,Z 358.747,A -85,B 0,C 180,E1 -21008.495,E2 -21008.495} C_VEL
LIN {X 0,Y 234.624,Z 343.734,A -85,B 0,C 180,E1 -21009.535,E2 -21009.535} C_VEL
LIN {X 0,Y 236.34,Z 328.105,A -85,B 0,C 180,E1 -21010.3,E2 -21010.3} C_VEL
LIN {X 0,Y 238.418,Z 291.335,A -85,B 0,C 180,E1 -21011.397,E2 -21011.397} C_VEL
LIN {X 0,Y 241.655,Z 230.298,A -85,B 0,C 180,E1 -21013.113,E2 -21013.113} C_VEL
LIN {X 0,Y 234.464,Z 212.01,A -85,B 0,C 180,E1 -21015.143,E2 -21015.143} C_VEL
LIN {X 0,Y 227.521,Z 196.665,A -85,B 0,C 180,E1 -21017.191,E2 -21017.191} C_VEL
LIN {X 0,Y 219.79,Z 181.824,A -85,B 0,C 180,E1 -21019.571,E2 -21019.571} C_VEL
LIN {X 0,Y 214.772,Z 173.149,A -85,B 0,C 180,E1 -21021.207,E2 -21021.207} C_VEL
LIN {X 0,Y 212.221,Z 169.232,A -85,B 0,C 180,E1 -21022.063,E2 -21022.063} C_VEL
LIN {X 0,Y 210.101,Z 166.075,A -85,B 0,C 180,E1 -21022.795,E2 -21022.795} C_VEL
LIN {X 0,Y 209.219,Z 164.918,A -85,B 0,C 180,E1 -21023.099,E2 -21023.099} C_VEL
LIN {X 0,Y 207.318,Z 162.5,A -85,B 0,C 180,E1 -21023.764,E2 -21023.764} C_VEL
LIN {X 0,Y 206.695,Z 160.36,A -85,B 0,C 180,E1 -21024.09,E2 -21024.09} C_VEL
LIN {X 0,Y 206.711,Z 160.358,A -85,B 0,C 180,E1 -21028.211,E2 -21028.211} C_VEL
LIN {X 0,Y 206.711,Z 160.323,A -85,B 0,C 180,E1 -21032.128,E2 -21032.128} C_VEL
LIN {X 0,Y 206.748,Z 160.354,A -85,B 0,C 180,E1 -21036.611,E2 -21036.611} C_VEL
LIN {X 0,Y 206.871,Z 160.331,A -85,B 0,C 180,E1 -21042.197,E2 -21042.197} C_VEL
LIN {X 0,Y 206.883,Z 160.338,A -85,B 0,C 180,E1 -21046.244,E2 -21046.244} C_VEL
LIN {X 0,Y 207.083,Z 160.316,A -85,B 0,C 180,E1 -21050.231,E2 -21050.231} C_VEL
LIN {X 0,Y 207.042,Z 160.318,A -85,B 0,C 180,E1 -21054.156,E2 -21054.156} C_VEL
LIN {X 0,Y 207.348,Z 160.242,A -85,B 0,C 180,E1 -21058.058,E2 -21058.058} C_VEL
LIN {X 0,Y 207.484,Z 160.217,A -85,B 0,C 180,E1 -21060.001,E2 -21060.001} C_VEL
LIN {X 0,Y 207.346,Z 160.256,A -85,B 0,C 180,E1 -21061.943,E2 -21061.943} C_VEL
LIN {X 0,Y 207.126,Z 160.27,A -85,B 0,C 180,E1 -21067.801,E2 -21067.801} C_VEL
LIN {X 0,Y 206.905,Z 160.306,A -85,B 0,C 180,E1 -21071.76,E2 -21071.76} C_VEL
LIN {X 0,Y 206.803,Z 160.343,A -85,B 0,C 180,E1 -21075.777,E2 -21075.777} C_VEL
LIN {X 0,Y 206.713,Z 160.36,A -85,B 0,C 180,E1 -21079.877,E2 -21079.877} C_VEL
LIN {X 0,Y 206.725,Z 160.36,A -85,B 0,C 180,E1 -21084.078,E2 -21084.078} C_VEL
LIN {X 0,Y 206.691,Z 160.322,A -85,B 0,C 180,E1 -21088.428,E2 -21088.428} C_VEL
LIN {X 0,Y 206.699,Z 160.356,A -85,B 0,C 180,E1 -21092.959,E2 -21092.959} C_VEL
LIN {X 0,Y 206.672,Z 160.327,A -85,B 0,C 180,E1 -21097.743,E2 -21097.743} C_VEL
LIN {X 0,Y 206.638,Z 160.367,A -85,B 0,C 180,E1 -21101.56,E2 -21101.56} C_VEL
LIN {X 0,Y 206.634,Z 160.34,A -85,B 0,C 180,E1 -21105.583,E2 -21105.583} C_VEL
LIN {X 0,Y 206.65,Z 160.368,A -85,B 0,C 180,E1 -21109.745,E2 -21109.745} C_VEL
LIN {X 0,Y 206.704,Z 160.361,A -85,B 0,C 180,E1 -21114.689,E2 -21114.689} C_VEL
LIN {X 0,Y 206.747,Z 160.563,A -85,B 0,C 180,E1 -21115.446,E2 -21115.446} C_VEL
LIN {X 0,Y 207.774,Z 163.278,A -85,B 0,C 180,E1 -21115.884,E2 -21115.884} C_VEL
LIN {X 0,Y 209.986,Z 165.823,A -85,B 0,C 180,E1 -21116.637,E2 -21116.637} C_VEL
LIN {X 0,Y 212.189,Z 169.2,A -85,B 0,C 180,E1 -21117.403,E2 -21117.403} C_VEL
LIN {X 0,Y 216.983,Z 176.278,A -85,B 0,C 180,E1 -21118.972,E2 -21118.972} C_VEL
LIN {X 0,Y 223.801,Z 186.871,A -85,B 0,C 180,E1 -21121.051,E2 -21121.051} C_VEL
LIN {X 0,Y 232.908,Z 202.641,A -85,B 0,C 180,E1 -21123.649,E2 -21123.649} C_VEL
LIN {X 0,Y 238.007,Z 212.902,A -85,B 0,C 180,E1 -21125.04,E2 -21125.04} C_VEL
LIN {X 0,Y 241.954,Z 222.58,A -85,B 0,C 180,E1 -21126.124,E2 -21126.124} C_VEL
LIN {X 0,Y 236.708,Z 316.376,A -85,B 0,C 180,E1 -21128.785,E2 -21128.785} C_VEL
LIN {X 0,Y 235.105,Z 332.037,A -85,B 0,C 180,E1 -21129.55,E2 -21129.55} C_VEL
LIN {X 0,Y 233.015,Z 347.039,A -85,B 0,C 180,E1 -21130.623,E2 -21130.623} C_VEL
LIN {X 0,Y 230.317,Z 361.596,A -85,B 0,C 180,E1 -21132.003,E2 -21132.003} C_VEL
LIN {X 0,Y 227.522,Z 374.836,A -85,B 0,C 180,E1 -21133.628,E2 -21133.628} C_VEL
LIN {X 0,Y 224.068,Z 388.384,A -85,B 0,C 180,E1 -21135.699,E2 -21135.699} C_VEL
LIN {X 0,Y 220.537,Z 400.703,A -85,B 0,C 180,E1 -21138.044,E2 -21138.044} C_VEL
LIN {X 0,Y 217.169,Z 411.915,A -85,B 0,C 180,E1 -21140.687,E2 -21140.687} C_VEL
LIN {X 0,Y 213.71,Z 422.804,A -85,B 0,C 180,E1 -21143.864,E2 -21143.864} C_VEL
LIN {X 0,Y 211.173,Z 430.999,A -85,B 0,C 180,E1 -21146.799,E2 -21146.799} C_VEL
LIN {X 0,Y 208.862,Z 438.356,A -85,B 0,C 180,E1 -21149.999,E2 -21149.999} C_VEL
LIN {X 0,Y 206.799,Z 445.572,A -85,B 0,C 180,E1 -21153.897,E2 -21153.897} C_VEL
LIN {X 0,Y 205.406,Z 451.256,A -85,B 0,C 180,E1 -21157.865,E2 -21157.865} C_VEL
LIN {X 0,Y 204.456,Z 455.567,A -85,B 0,C 180,E1 -21161.902,E2 -21161.902} C_VEL
LIN {X 0,Y 204.032,Z 458.585,A -85,B 0,C 180,E1 -21165.995,E2 -21165.995} C_VEL
LIN {X 0,Y 203.98,Z 460.361,A -85,B 0,C 180,E1 -21170.153,E2 -21170.153} C_VEL
LIN {X 0,Y 204.103,Z 460.782,A -85,B 0,C 180,E1 -21172.257,E2 -21172.257} C_VEL
LIN {X 0,Y 204.742,Z 460.671,A -85,B 0,C 180,E1 -21176.502,E2 -21176.502} C_VEL
LIN {X 0,Y 206.008,Z 459.25,A -85,B 0,C 180,E1 -21180.778,E2 -21180.778} C_VEL
LIN {X 0,Y 208.065,Z 456.453,A -85,B 0,C 180,E1 -21185.044,E2 -21185.044} C_VEL
LIN {X 0,Y 211.109,Z 452.188,A -85,B 0,C 180,E1 -21189.236,E2 -21189.236} C_VEL
LIN {X 0,Y 215.06,Z 446.322,A -85,B 0,C 180,E1 -21193.334,E2 -21193.334} C_VEL
LIN {X 0,Y 219.361,Z 439.764,A -85,B 0,C 180,E1 -21196.791,E2 -21196.791} C_VEL
LIN {X 0,Y 224.337,Z 431.626,A -85,B 0,C 180,E1 -21200.132,E2 -21200.132} C_VEL
LIN {X 0,Y 229.238,Z 423.228,A -85,B 0,C 180,E1 -21202.854,E2 -21202.854} C_VEL
LIN {X 0,Y 235.03,Z 412.357,A -85,B 0,C 180,E1 -21205.666,E2 -21205.666} C_VEL
LIN {X 0,Y 240.394,Z 401.156,A -85,B 0,C 180,E1 -21207.975,E2 -21207.975} C_VEL
LIN {X 0,Y 245.588,Z 389.067,A -85,B 0,C 180,E1 -21209.958,E2 -21209.958} C_VEL
LIN {X 0,Y 250.313,Z 376.365,A -85,B 0,C 180,E1 -21211.628,E2 -21211.628} C_VEL
LIN {X 0,Y 254.415,Z 363.398,A -85,B 0,C 180,E1 -21212.983,E2 -21212.983} C_VEL
LIN {X 0,Y 257.897,Z 350.192,A -85,B 0,C 180,E1 -21214.064,E2 -21214.064} C_VEL
LIN {X 0,Y 260.671,Z 336.843,A -85,B 0,C 180,E1 -21214.919,E2 -21214.919} C_VEL
LIN {X 0,Y 263.114,Z 321.295,A -85,B 0,C 180,E1 -21215.613,E2 -21215.613} C_VEL
LIN {X 0,Y 264.703,Z 304.152,A -85,B 0,C 180,E1 -21216.121,E2 -21216.121} C_VEL
LIN {X 0,Y 269.192,Z 241.914,A -85,B 0,C 180,E1 -21217.704,E2 -21217.704} C_VEL
LIN {X 0,Y 263.679,Z 230.756,A -85,B 0,C 180,E1 -21220.102,E2 -21220.102} C_VEL
LIN {X 0,Y 259.466,Z 223.717,A -85,B 0,C 180,E1 -21222.042,E2 -21222.042} C_VEL
LIN {X 0,Y 254.725,Z 216.478,A -85,B 0,C 180,E1 -21224.483,E2 -21224.483} C_VEL
LIN {X 0,Y 251.551,Z 211.887,A -85,B 0,C 180,E1 -21226.281,E2 -21226.281} C_VEL
LIN {X 0,Y 249.795,Z 209.352,A -85,B 0,C 180,E1 -21227.35,E2 -21227.35} C_VEL
LIN {X 0,Y 246.643,Z 205.025,A -85,B 0,C 180,E1 -21229.42,E2 -21229.42} C_VEL
LIN {X 0,Y 243.887,Z 201.071,A -85,B 0,C 180,E1 -21231.506,E2 -21231.506} C_VEL
LIN {X 0,Y 241.006,Z 197.398,A -85,B 0,C 180,E1 -21234.01,E2 -21234.01} C_VEL
LIN {X 0,Y 240.064,Z 195.925,A -85,B 0,C 180,E1 -21234.961,E2 -21234.961} C_VEL
LIN {X 0,Y 237.577,Z 193.639,A -85,B 0,C 180,E1 -21237.625,E2 -21237.625} C_VEL
LIN {X 0,Y 236.174,Z 190.581,A -85,B 0,C 180,E1 -21239.786,E2 -21239.786} C_VEL
LIN {X 0,Y 232.995,Z 188.171,A -85,B 0,C 180,E1 -21248.674,E2 -21248.674} C_VEL
LIN {X 0,Y 233.809,Z 189.425,A -85,B 0,C 180,E1 -21254.358,E2 -21254.358} C_VEL
LIN {X 0,Y 236.034,Z 191.011,A -85,B 0,C 180,E1 -21258.759,E2 -21258.759} C_VEL
LIN {X 0,Y 237.524,Z 193.916,A -85,B 0,C 180,E1 -21261.016,E2 -21261.016} C_VEL
LIN {X 0,Y 238.007,Z 194.5,A -85,B 0,C 180,E1 -21261.599,E2 -21261.599} C_VEL
LIN {X 0,Y 239.082,Z 196.55,A -85,B 0,C 180,E1 -21262.898,E2 -21262.898} C_VEL
LIN {X 0,Y 240.017,Z 199.679,A -85,B 0,C 180,E1 -21264.083,E2 -21264.083} C_VEL
LIN {X 0,Y 242.648,Z 209.335,A -85,B 0,C 180,E1 -21267.065,E2 -21267.065} C_VEL
LIN {X 0,Y 243.583,Z 211.253,A -85,B 0,C 180,E1 -21267.865,E2 -21267.865} C_VEL
LIN {X 0,Y 246.774,Z 216.264,A -85,B 0,C 180,E1 -21270.191,E2 -21270.191} C_VEL
LIN {X 0,Y 250.464,Z 222.674,A -85,B 0,C 180,E1 -21272.585,E2 -21272.585} C_VEL
LIN {X 0,Y 253.854,Z 228.711,A -85,B 0,C 180,E1 -21274.564,E2 -21274.564} C_VEL
LIN {X 0,Y 258.717,Z 238.352,A -85,B 0,C 180,E1 -21277.151,E2 -21277.151} C_VEL
LIN {X 0,Y 263.946,Z 249.671,A -85,B 0,C 180,E1 -21279.627,E2 -21279.627} C_VEL
LIN {X 0,Y 264.637,Z 251.486,A -85,B 0,C 180,E1 -21279.951,E2 -21279.951} C_VEL
LIN {X 0,Y 259.01,Z 325.262,A -85,B 0,C 180,E1 -21281.86,E2 -21281.86} C_VEL
LIN {X 0,Y 256.638,Z 341.203,A -85,B 0,C 180,E1 -21282.467,E2 -21282.467} C_VEL
LIN {X 0,Y 253.429,Z 356.165,A -85,B 0,C 180,E1 -21283.285,E2 -21283.285} C_VEL
LIN {X 0,Y 249.42,Z 370.631,A -85,B 0,C 180,E1 -21284.357,E2 -21284.357} C_VEL
LIN {X 0,Y 245.087,Z 383.764,A -85,B 0,C 180,E1 -21285.657,E2 -21285.657} C_VEL
LIN {X 0,Y 240.118,Z 396.362,A -85,B 0,C 180,E1 -21287.206,E2 -21287.206} C_VEL
LIN {X 0,Y 235.308,Z 407.364,A -85,B 0,C 180,E1 -21288.923,E2 -21288.923} C_VEL
LIN {X 0,Y 229.628,Z 418.907,A -85,B 0,C 180,E1 -21291.14,E2 -21291.14} C_VEL
LIN {X 0,Y 224.351,Z 428.669,A -85,B 0,C 180,E1 -21293.474,E2 -21293.474} C_VEL
LIN {X 0,Y 218.624,Z 438.28,A -85,B 0,C 180,E1 -21296.323,E2 -21296.323} C_VEL
LIN {X 0,Y 214.321,Z 445.263,A -85,B 0,C 180,E1 -21298.905,E2 -21298.905} C_VEL
LIN {X 0,Y 209.858,Z 452.148,A -85,B 0,C 180,E1 -21302.041,E2 -21302.041} C_VEL
LIN {X 0,Y 205.609,Z 458.582,A -85,B 0,C 180,E1 -21305.785,E2 -21305.785} C_VEL
LIN {X 0,Y 201.763,Z 464.171,A -85,B 0,C 180,E1 -21310.132,E2 -21310.132} C_VEL
LIN {X 0,Y 199.778,Z 467.469,A -85,B 0,C 180,E1 -21313.655,E2 -21313.655} C_VEL
LIN {X 0,Y 198.16,Z 470.094,A -85,B 0,C 180,E1 -21317.714,E2 -21317.714} C_VEL
LIN {X 0,Y 197.386,Z 471.549,A -85,B 0,C 180,E1 -21321.813,E2 -21321.813} C_VEL
LIN {X 0,Y 197.164,Z 471.871,A -85,B 0,C 180,E1 -21326.431,E2 -21326.431} C_VEL
LIN {X 0,Y 197.396,Z 471.14,A -85,B 0,C 180,E1 -21330.001,E2 -21330.001} C_VEL
LIN {X 0,Y 197.283,Z 469.183,A -85,B 0,C 180,E1 -21334.086,E2 -21334.086} C_VEL
LIN {X 0,Y 197.412,Z 465.944,A -85,B 0,C 180,E1 -21338.188,E2 -21338.188} C_VEL
LIN {X 0,Y 197.996,Z 461.379,A -85,B 0,C 180,E1 -21342.298,E2 -21342.298} C_VEL
LIN {X 0,Y 199.33,Z 455.383,A -85,B 0,C 180,E1 -21346.384,E2 -21346.384} C_VEL
LIN {X 0,Y 201.179,Z 448.803,A -85,B 0,C 180,E1 -21349.926,E2 -21349.926} C_VEL
LIN {X 0,Y 203.593,Z 440.882,A -85,B 0,C 180,E1 -21353.39,E2 -21353.39} C_VEL
LIN {X 0,Y 206.773,Z 431.314,A -85,B 0,C 180,E1 -21356.767,E2 -21356.767} C_VEL
LIN {X 0,Y 210.139,Z 420.803,A -85,B 0,C 180,E1 -21359.778,E2 -21359.778} C_VEL
LIN {X 0,Y 213.884,Z 408.781,A -85,B 0,C 180,E1 -21362.553,E2 -21362.553} C_VEL
LIN {X 0,Y 217.289,Z 397.002,A -85,B 0,C 180,E1 -21364.756,E2 -21364.756} C_VEL
LIN {X 0,Y 220.763,Z 384.334,A -85,B 0,C 180,E1 -21366.65,E2 -21366.65} C_VEL
LIN {X 0,Y 223.974,Z 370.289,A -85,B 0,C 180,E1 -21368.33,E2 -21368.33} C_VEL
LIN {X 0,Y 226.646,Z 356.422,A -85,B 0,C 180,E1 -21369.615,E2 -21369.615} C_VEL
LIN {X 0,Y 229,Z 341.422,A -85,B 0,C 180,E1 -21370.633,E2 -21370.633} C_VEL
LIN {X 0,Y 230.639,Z 325.862,A -85,B 0,C 180,E1 -21371.367,E2 -21371.367} C_VEL
LIN {X 0,Y 235.888,Z 232.212,A -85,B 0,C 180,E1 -21374.081,E2 -21374.081} C_VEL
LIN {X 0,Y 228.764,Z 213.993,A -85,B 0,C 180,E1 -21376.206,E2 -21376.206} C_VEL
LIN {X 0,Y 222.259,Z 199.59,A -85,B 0,C 180,E1 -21378.222,E2 -21378.222} C_VEL
LIN {X 0,Y 213.894,Z 183.478,A -85,B 0,C 180,E1 -21380.946,E2 -21380.946} C_VEL
LIN {X 0,Y 208.388,Z 174.512,A -85,B 0,C 180,E1 -21382.851,E2 -21382.851} C_VEL
LIN {X 0,Y 205.438,Z 170.322,A -85,B 0,C 180,E1 -21383.911,E2 -21383.911} C_VEL
LIN {X 0,Y 203.271,Z 167.214,A -85,B 0,C 180,E1 -21384.724,E2 -21384.724} C_VEL
LIN {X 0,Y 202.55,Z 166.133,A -85,B 0,C 180,E1 -21385.004,E2 -21385.004} C_VEL
LIN {X 0,Y 200.527,Z 163.941,A -85,B 0,C 180,E1 -21385.755,E2 -21385.755} C_VEL
LIN {X 0,Y 199.616,Z 161.243,A -85,B 0,C 180,E1 -21386.249,E2 -21386.249} C_VEL
LIN {X 0,Y 199.688,Z 161.232,A -85,B 0,C 180,E1 -21388.136,E2 -21388.136} C_VEL
LIN {X 0,Y 199.645,Z 161.203,A -85,B 0,C 180,E1 -21392.766,E2 -21392.766} C_VEL
LIN {X 0,Y 199.71,Z 161.226,A -85,B 0,C 180,E1 -21397.227,E2 -21397.227} C_VEL
LIN {X 0,Y 199.798,Z 161.216,A -85,B 0,C 180,E1 -21401.76,E2 -21401.76} C_VEL
LIN {X 0,Y 199.823,Z 161.22,A -85,B 0,C 180,E1 -21405.748,E2 -21405.748} C_VEL
LIN {X 0,Y 200.027,Z 161.194,A -85,B 0,C 180,E1 -21409.883,E2 -21409.883} C_VEL
LIN {X 0,Y 200.006,Z 161.193,A -85,B 0,C 180,E1 -21413.95,E2 -21413.95} C_VEL
LIN {X 0,Y 200.291,Z 161.121,A -85,B 0,C 180,E1 -21417.99,E2 -21417.99} C_VEL
LIN {X 0,Y 200.451,Z 161.092,A -85,B 0,C 180,E1 -21420.001,E2 -21420.001} C_VEL
LIN {X 0,Y 199.989,Z 161.196,A -85,B 0,C 180,E1 -21424.031,E2 -21424.031} C_VEL
LIN {X 0,Y 200.074,Z 161.144,A -85,B 0,C 180,E1 -21428.078,E2 -21428.078} C_VEL
LIN {X 0,Y 199.855,Z 161.19,A -85,B 0,C 180,E1 -21432.181,E2 -21432.181} C_VEL
LIN {X 0,Y 199.744,Z 161.218,A -85,B 0,C 180,E1 -21436.35,E2 -21436.35} C_VEL
LIN {X 0,Y 199.646,Z 161.238,A -85,B 0,C 180,E1 -21440.612,E2 -21440.612} C_VEL
LIN {X 0,Y 199.639,Z 161.243,A -85,B 0,C 180,E1 -21444.99,E2 -21444.99} C_VEL
LIN {X 0,Y 199.611,Z 161.199,A -85,B 0,C 180,E1 -21449.534,E2 -21449.534} C_VEL
LIN {X 0,Y 199.67,Z 161.222,A -85,B 0,C 180,E1 -21452.352,E2 -21452.352} C_VEL
LIN {X 0,Y 199.622,Z 161.212,A -85,B 0,C 180,E1 -21456.765,E2 -21456.765} C_VEL
LIN {X 0,Y 199.599,Z 161.211,A -85,B 0,C 180,E1 -21459.331,E2 -21459.331} C_VEL
LIN {X 0,Y 199.573,Z 161.25,A -85,B 0,C 180,E1 -21462.308,E2 -21462.308} C_VEL
LIN {X 0,Y 199.58,Z 161.219,A -85,B 0,C 180,E1 -21465.227,E2 -21465.227} C_VEL
LIN {X 0,Y 199.573,Z 161.237,A -85,B 0,C 180,E1 -21468.002,E2 -21468.002} C_VEL
LIN {X 0,Y 199.6,Z 161.232,A -85,B 0,C 180,E1 -21470.773,E2 -21470.773} C_VEL
LIN {X 0,Y 199.636,Z 161.42,A -85,B 0,C 180,E1 -21473.298,E2 -21473.298} C_VEL
LIN {X 0,Y 200.521,Z 163.945,A -85,B 0,C 180,E1 -21473.72,E2 -21473.72} C_VEL
LIN {X 0,Y 202.655,Z 166.172,A -85,B 0,C 180,E1 -21474.507,E2 -21474.507} C_VEL
LIN {X 0,Y 205.304,Z 170.172,A -85,B 0,C 180,E1 -21475.518,E2 -21475.518} C_VEL
LIN {X 0,Y 206.555,Z 171.854,A -85,B 0,C 180,E1 -21475.97,E2 -21475.97} C_VEL
LIN {X 0,Y 214.411,Z 183.449,A -85,B 0,C 180,E1 -21478.662,E2 -21478.662} C_VEL
LIN {X 0,Y 222.702,Z 197.032,A -85,B 0,C 180,E1 -21481.245,E2 -21481.245} C_VEL
LIN {X 0,Y 230.332,Z 210.974,A -85,B 0,C 180,E1 -21483.465,E2 -21483.465} C_VEL
LIN {X 0,Y 234.333,Z 219.864,A -85,B 0,C 180,E1 -21484.614,E2 -21484.614} C_VEL
LIN {X 0,Y 236.151,Z 224.518,A -85,B 0,C 180,E1 -21485.142,E2 -21485.142} C_VEL
LIN {X 0,Y 230.865,Z 316.595,A -85,B 0,C 180,E1 -21487.81,E2 -21487.81} C_VEL
LIN {X 0,Y 229.198,Z 332.255,A -85,B 0,C 180,E1 -21488.586,E2 -21488.586} C_VEL
LIN {X 0,Y 227.113,Z 346.699,A -85,B 0,C 180,E1 -21489.626,E2 -21489.626} C_VEL
LIN {X 0,Y 224.336,Z 361.364,A -85,B 0,C 180,E1 -21491.032,E2 -21491.032} C_VEL
LIN {X 0,Y 221.431,Z 374.67,A -85,B 0,C 180,E1 -21492.688,E2 -21492.688} C_VEL
LIN {X 0,Y 217.852,Z 388.29,A -85,B 0,C 180,E1 -21494.803,E2 -21494.803} C_VEL
LIN {X 0,Y 214.179,Z 400.66,A -85,B 0,C 180,E1 -21497.202,E2 -21497.202} C_VEL
LIN {X 0,Y 210.671,Z 411.907,A -85,B 0,C 180,E1 -21499.912,E2 -21499.912} C_VEL
LIN {X 0,Y 207.079,Z 422.833,A -85,B 0,C 180,E1 -21503.177,E2 -21503.177} C_VEL
LIN {X 0,Y 204.209,Z 431.66,A -85,B 0,C 180,E1 -21506.442,E2 -21506.442} C_VEL
LIN {X 0,Y 201.686,Z 439.454,A -85,B 0,C 180,E1 -21509.999,E2 -21509.999} C_VEL
LIN {X 0,Y 199.611,Z 446.495,A -85,B 0,C 180,E1 -21514.037,E2 -21514.037} C_VEL
LIN {X 0,Y 198.226,Z 452.017,A -85,B 0,C 180,E1 -21518.152,E2 -21518.152} C_VEL
LIN {X 0,Y 197.277,Z 456.178,A -85,B 0,C 180,E1 -21522.341,E2 -21522.341} C_VEL
LIN {X 0,Y 196.883,Z 459.051,A -85,B 0,C 180,E1 -21526.592,E2 -21526.592} C_VEL
LIN {X 0,Y 196.922,Z 460.682,A -85,B 0,C 180,E1 -21530.909,E2 -21530.909} C_VEL
LIN {X 0,Y 197.374,Z 461.061,A -85,B 0,C 180,E1 -21535.295,E2 -21535.295} C_VEL
LIN {X 0,Y 198.485,Z 460.148,A -85,B 0,C 180,E1 -21539.716,E2 -21539.716} C_VEL
LIN {X 0,Y 200.402,Z 457.89,A -85,B 0,C 180,E1 -21544.132,E2 -21544.132} C_VEL
LIN {X 0,Y 203.276,Z 454.205,A -85,B 0,C 180,E1 -21548.485,E2 -21548.485} C_VEL
LIN {X 0,Y 207.088,Z 448.979,A -85,B 0,C 180,E1 -21552.745,E2 -21552.745} C_VEL
LIN {X 0,Y 210.85,Z 443.671,A -85,B 0,C 180,E1 -21556.015,E2 -21556.015} C_VEL
LIN {X 0,Y 215.373,Z 436.941,A -85,B 0,C 180,E1 -21559.258,E2 -21559.258} C_VEL
LIN {X 0,Y 221.052,Z 427.983,A -85,B 0,C 180,E1 -21562.639,E2 -21562.639} C_VEL
LIN {X 0,Y 226.442,Z 418.859,A -85,B 0,C 180,E1 -21565.332,E2 -21565.332} C_VEL
LIN {X 0,Y 232.233,Z 407.955,A -85,B 0,C 180,E1 -21567.924,E2 -21567.924} C_VEL
LIN {X 0,Y 237.772,Z 396.408,A -85,B 0,C 180,E1 -21570.09,E2 -21570.09} C_VEL
LIN {X 0,Y 242.937,Z 384.166,A -85,B 0,C 180,E1 -21571.925,E2 -21571.925} C_VEL
LIN {X 0,Y 247.465,Z 371.552,A -85,B 0,C 180,E1 -21573.456,E2 -21573.456} C_VEL
LIN {X 0,Y 251.438,Z 358.546,A -85,B 0,C 180,E1 -21574.701,E2 -21574.701} C_VEL
LIN {X 0,Y 255.161,Z 343.24,A -85,B 0,C 180,E1 -21575.835,E2 -21575.835} C_VEL
LIN {X 0,Y 257.964,Z 328.424,A -85,B 0,C 180,E1 -21576.604,E2 -21576.604} C_VEL
LIN {X 0,Y 259.865,Z 313.298,A -85,B 0,C 180,E1 -21577.148,E2 -21577.148} C_VEL
LIN {X 0,Y 265.108,Z 245.137,A -85,B 0,C 180,E1 -21578.87,E2 -21578.87} C_VEL
LIN {X 0,Y 259.613,Z 234.056,A -85,B 0,C 180,E1 -21581.406,E2 -21581.406} C_VEL
LIN {X 0,Y 254.556,Z 225.79,A -85,B 0,C 180,E1 -21583.972,E2 -21583.972} C_VEL
LIN {X 0,Y 250.054,Z 218.975,A -85,B 0,C 180,E1 -21586.536,E2 -21586.536} C_VEL
LIN {X 0,Y 247.671,Z 215.514,A -85,B 0,C 180,E1 -21588.031,E2 -21588.031} C_VEL
LIN {X 0,Y 244.98,Z 211.652,A -85,B 0,C 180,E1 -21589.874,E2 -21589.874} C_VEL
LIN {X 0,Y 241.867,Z 207.206,A -85,B 0,C 180,E1 -21592.355,E2 -21592.355} C_VEL
LIN {X 0,Y 239.125,Z 203.272,A -85,B 0,C 180,E1 -21594.941,E2 -21594.941} C_VEL
LIN {X 0,Y 236.075,Z 200.017,A -85,B 0,C 180,E1 -21598.383,E2 -21598.383} C_VEL
LIN {X 0,Y 234.86,Z 197.419,A -85,B 0,C 180,E1 -21600.379,E2 -21600.379} C_VEL
LIN {X 0,Y 232.098,Z 195.22,A -85,B 0,C 180,E1 -21608.707,E2 -21608.707} C_VEL
LIN {X 0,Y 233.092,Z 196.623,A -85,B 0,C 180,E1 -21614.849,E2 -21614.849} C_VEL
LIN {X 0,Y 234.85,Z 197.843,A -85,B 0,C 180,E1 -21618.342,E2 -21618.342} C_VEL
LIN {X 0,Y 236.495,Z 200.98,A -85,B 0,C 180,E1 -21620.891,E2 -21620.891} C_VEL
LIN {X 0,Y 238.544,Z 203.267,A -85,B 0,C 180,E1 -21623.206,E2 -21623.206} C_VEL
LIN {X 0,Y 240.028,Z 205.5,A -85,B 0,C 180,E1 -21624.724,E2 -21624.724} C_VEL
LIN {X 0,Y 243.256,Z 210.63,A -85,B 0,C 180,E1 -21627.595,E2 -21627.595} C_VEL
LIN {X 0,Y 243.583,Z 211.253,A -85,B 0,C 180,E1 -21627.865,E2 -21627.865} C_VEL
LIN {X 0,Y 244.968,Z 214.353,A -85,B 0,C 180,E1 -21628.996,E2 -21628.996} C_VEL
LIN {X 0,Y 246.852,Z 221.189,A -85,B 0,C 180,E1 -21630.607,E2 -21630.607} C_VEL
LIN {X 0,Y 249.211,Z 229.851,A -85,B 0,C 180,E1 -21632.46,E2 -21632.46} C_VEL
LIN {X 0,Y 250.256,Z 232.329,A -85,B 0,C 180,E1 -21633.139,E2 -21633.139} C_VEL
LIN {X 0,Y 255.185,Z 242.233,A -85,B 0,C 180,E1 -21635.968,E2 -21635.968} C_VEL
LIN {X 0,Y 260.224,Z 253.483,A -85,B 0,C 180,E1 -21638.532,E2 -21638.532} C_VEL
LIN {X 0,Y 260.635,Z 254.417,A -85,B 0,C 180,E1 -21638.727,E2 -21638.727} C_VEL
LIN {X 0,Y 254.98,Z 325.469,A -85,B 0,C 180,E1 -21640.563,E2 -21640.563} C_VEL
LIN {X 0,Y 252.596,Z 340.992,A -85,B 0,C 180,E1 -21641.153,E2 -21641.153} C_VEL
LIN {X 0,Y 249.285,Z 355.961,A -85,B 0,C 180,E1 -21641.963,E2 -21641.963} C_VEL
LIN {X 0,Y 245.15,Z 370.432,A -85,B 0,C 180,E1 -21643.027,E2 -21643.027} C_VEL
LIN {X 0,Y 240.687,Z 383.564,A -85,B 0,C 180,E1 -21644.325,E2 -21644.325} C_VEL
LIN {X 0,Y 235.596,Z 396.042,A -85,B 0,C 180,E1 -21645.854,E2 -21645.854} C_VEL
LIN {X 0,Y 230.582,Z 407.163,A -85,B 0,C 180,E1 -21647.597,E2 -21647.597} C_VEL
LIN {X 0,Y 225.17,Z 417.826,A -85,B 0,C 180,E1 -21649.636,E2 -21649.636} C_VEL
LIN {X 0,Y 219.593,Z 427.739,A -85,B 0,C 180,E1 -21651.97,E2 -21651.97} C_VEL
LIN {X 0,Y 213.559,Z 437.474,A -85,B 0,C 180,E1 -21654.838,E2 -21654.838} C_VEL
LIN {X 0,Y 208.242,Z 445.608,A -85,B 0,C 180,E1 -21657.891,E2 -21657.891} C_VEL
LIN {X 0,Y 203.6,Z 452.367,A -85,B 0,C 180,E1 -21661.102,E2 -21661.102} C_VEL
LIN {X 0,Y 199.106,Z 458.703,A -85,B 0,C 180,E1 -21664.94,E2 -21664.94} C_VEL
LIN {X 0,Y 195.471,Z 463.688,A -85,B 0,C 180,E1 -21668.929,E2 -21668.929} C_VEL
LIN {X 0,Y 192.902,Z 467.432,A -85,B 0,C 180,E1 -21673.055,E2 -21673.055} C_VEL
LIN {X 0,Y 191.165,Z 470.009,A -85,B 0,C 180,E1 -21677.257,E2 -21677.257} C_VEL
LIN {X 0,Y 190.325,Z 471.403,A -85,B 0,C 180,E1 -21681.507,E2 -21681.507} C_VEL
LIN {X 0,Y 190.08,Z 471.685,A -85,B 0,C 180,E1 -21685.76,E2 -21685.76} C_VEL
LIN {X 0,Y 190.315,Z 470.85,A -85,B 0,C 180,E1 -21690.001,E2 -21690.001} C_VEL
LIN {X 0,Y 190.193,Z 468.823,A -85,B 0,C 180,E1 -21694.239,E2 -21694.239} C_VEL
LIN {X 0,Y 190.347,Z 465.538,A -85,B 0,C 180,E1 -21698.494,E2 -21698.494} C_VEL
LIN {X 0,Y 191,Z 460.893,A -85,B 0,C 180,E1 -21702.755,E2 -21702.755} C_VEL
LIN {X 0,Y 192.444,Z 454.81,A -85,B 0,C 180,E1 -21706.988,E2 -21706.988} C_VEL
LIN {X 0,Y 194.736,Z 447.125,A -85,B 0,C 180,E1 -21711.156,E2 -21711.156} C_VEL
LIN {X 0,Y 197.436,Z 438.853,A -85,B 0,C 180,E1 -21714.726,E2 -21714.726} C_VEL
LIN {X 0,Y 200.339,Z 430.422,A -85,B 0,C 180,E1 -21717.699,E2 -21717.699} C_VEL
LIN {X 0,Y 203.812,Z 420.032,A -85,B 0,C 180,E1 -21720.72,E2 -21720.72} C_VEL
LIN {X 0,Y 207.861,Z 407.593,A -85,B 0,C 180,E1 -21723.619,E2 -21723.619} C_VEL
LIN {X 0,Y 211.039,Z 396.922,A -85,B 0,C 180,E1 -21725.648,E2 -21725.648} C_VEL
LIN {X 0,Y 214.618,Z 384.277,A -85,B 0,C 180,E1 -21727.584,E2 -21727.584} C_VEL
LIN {X 0,Y 217.881,Z 370.504,A -85,B 0,C 180,E1 -21729.273,E2 -21729.273} C_VEL
LIN {X 0,Y 220.705,Z 356.454,A -85,B 0,C 180,E1 -21730.603,E2 -21730.603} C_VEL
LIN {X 0,Y 223.239,Z 340.627,A -85,B 0,C 180,E1 -21731.688,E2 -21731.688} C_VEL
LIN {X 0,Y 224.92,Z 324.682,A -85,B 0,C 180,E1 -21732.435,E2 -21732.435} C_VEL
LIN {X 0,Y 230.125,Z 233.964,A -85,B 0,C 180,E1 -21735.117,E2 -21735.117} C_VEL
LIN {X 0,Y 222.854,Z 215.297,A -85,B 0,C 180,E1 -21737.416,E2 -21737.416} C_VEL
LIN {X 0,Y 216.173,Z 200.827,A -85,B 0,C 180,E1 -21739.577,E2 -21739.577} C_VEL
LIN {X 0,Y 209.242,Z 187.483,A -85,B 0,C 180,E1 -21741.974,E2 -21741.974} C_VEL
LIN {X 0,Y 204.746,Z 179.936,A -85,B 0,C 180,E1 -21743.617,E2 -21743.617} C_VEL
LIN {X 0,Y 198.726,Z 171.472,A -85,B 0,C 180,E1 -21745.923,E2 -21745.923} C_VEL
LIN {X 0,Y 196.481,Z 168.426,A -85,B 0,C 180,E1 -21746.831,E2 -21746.831} C_VEL
LIN {X 0,Y 195.717,Z 167.147,A -85,B 0,C 180,E1 -21747.162,E2 -21747.162} C_VEL
LIN {X 0,Y 193.586,Z 164.87,A -85,B 0,C 180,E1 -21748.037,E2 -21748.037} C_VEL
LIN {X 0,Y 192.617,Z 162.116,A -85,B 0,C 180,E1 -21748.596,E2 -21748.596} C_VEL
LIN {X 0,Y 192.622,Z 162.079,A -85,B 0,C 180,E1 -21751.686,E2 -21751.686} C_VEL
LIN {X 0,Y 192.681,Z 162.107,A -85,B 0,C 180,E1 -21756.346,E2 -21756.346} C_VEL
LIN {X 0,Y 192.733,Z 162.098,A -85,B 0,C 180,E1 -21761.461,E2 -21761.461} C_VEL
LIN {X 0,Y 192.752,Z 162.101,A -85,B 0,C 180,E1 -21765.214,E2 -21765.214} C_VEL
LIN {X 0,Y 192.949,Z 162.075,A -85,B 0,C 180,E1 -21769.568,E2 -21769.568} C_VEL
LIN {X 0,Y 192.97,Z 162.069,A -85,B 0,C 180,E1 -21773.728,E2 -21773.728} C_VEL
LIN {X 0,Y 193.235,Z 162,A -85,B 0,C 180,E1 -21777.917,E2 -21777.917} C_VEL
LIN {X 0,Y 193.417,Z 161.968,A -85,B 0,C 180,E1 -21780.001,E2 -21780.001} C_VEL
LIN {X 0,Y 192.936,Z 162.075,A -85,B 0,C 180,E1 -21784.179,E2 -21784.179} C_VEL
LIN {X 0,Y 193.026,Z 162.018,A -85,B 0,C 180,E1 -21788.375,E2 -21788.375} C_VEL
LIN {X 0,Y 192.782,Z 162.078,A -85,B 0,C 180,E1 -21792.636,E2 -21792.636} C_VEL
LIN {X 0,Y 192.687,Z 162.095,A -85,B 0,C 180,E1 -21796.966,E2 -21796.966} C_VEL
LIN {X 0,Y 192.58,Z 162.111,A -85,B 0,C 180,E1 -21801.405,E2 -21801.405} C_VEL
LIN {X 0,Y 192.63,Z 162.116,A -85,B 0,C 180,E1 -21804.199,E2 -21804.199} C_VEL
LIN {X 0,Y 192.605,Z 162.072,A -85,B 0,C 180,E1 -21808.865,E2 -21808.865} C_VEL
LIN {X 0,Y 192.599,Z 162.114,A -85,B 0,C 180,E1 -21813.187,E2 -21813.187} C_VEL
LIN {X 0,Y 192.546,Z 162.084,A -85,B 0,C 180,E1 -21818.354,E2 -21818.354} C_VEL
LIN {X 0,Y 192.491,Z 162.127,A -85,B 0,C 180,E1 -21823.094,E2 -21823.094} C_VEL
LIN {X 0,Y 192.488,Z 162.105,A -85,B 0,C 180,E1 -21826.907,E2 -21826.907} C_VEL
LIN {X 0,Y 192.573,Z 162.263,A -85,B 0,C 180,E1 -21830.913,E2 -21830.913} C_VEL
LIN {X 0,Y 193.501,Z 164.915,A -85,B 0,C 180,E1 -21831.403,E2 -21831.403} C_VEL
LIN {X 0,Y 195.553,Z 167.083,A -85,B 0,C 180,E1 -21832.249,E2 -21832.249} C_VEL
LIN {X 0,Y 196.302,Z 168.042,A -85,B 0,C 180,E1 -21832.559,E2 -21832.559} C_VEL
LIN {X 0,Y 198.517,Z 171.3,A -85,B 0,C 180,E1 -21833.476,E2 -21833.476} C_VEL
LIN {X 0,Y 199.705,Z 172.71,A -85,B 0,C 180,E1 -21833.935,E2 -21833.935} C_VEL
LIN {X 0,Y 205.99,Z 181.831,A -85,B 0,C 180,E1 -21836.317,E2 -21836.317} C_VEL
LIN {X 0,Y 213.741,Z 193.903,A -85,B 0,C 180,E1 -21838.984,E2 -21838.984} C_VEL
LIN {X 0,Y 222.214,Z 208.787,A -85,B 0,C 180,E1 -21841.644,E2 -21841.644} C_VEL
LIN {X 0,Y 227.679,Z 219.609,A -85,B 0,C 180,E1 -21843.273,E2 -21843.273} C_VEL
LIN {X 0,Y 230.432,Z 226.405,A -85,B 0,C 180,E1 -21844.111,E2 -21844.111} C_VEL
LIN {X 0,Y 225.087,Z 316.82,A -85,B 0,C 180,E1 -21846.783,E2 -21846.783} C_VEL
LIN {X 0,Y 223.36,Z 332.472,A -85,B 0,C 180,E1 -21847.572,E2 -21847.572} C_VEL
LIN {X 0,Y 221.089,Z 347.479,A -85,B 0,C 180,E1 -21848.679,E2 -21848.679} C_VEL
LIN {X 0,Y 218.442,Z 361.11,A -85,B 0,C 180,E1 -21850.01,E2 -21850.01} C_VEL
LIN {X 0,Y 215.129,Z 375.573,A -85,B 0,C 180,E1 -21851.85,E2 -21851.85} C_VEL
LIN {X 0,Y 211.399,Z 389.151,A -85,B 0,C 180,E1 -21854.031,E2 -21854.031} C_VEL
LIN {X 0,Y 207.883,Z 400.608,A -85,B 0,C 180,E1 -21856.31,E2 -21856.31} C_VEL
LIN {X 0,Y 204.229,Z 411.891,A -85,B 0,C 180,E1 -21859.089,E2 -21859.089} C_VEL
LIN {X 0,Y 200.462,Z 422.866,A -85,B 0,C 180,E1 -21862.445,E2 -21862.445} C_VEL
LIN {X 0,Y 197.253,Z 432.3,A -85,B 0,C 180,E1 -21866.063,E2 -21866.063} C_VEL
LIN {X 0,Y 194.487,Z 440.5,A -85,B 0,C 180,E1 -21869.999,E2 -21869.999} C_VEL
LIN {X 0,Y 192.42,Z 447.358,A -85,B 0,C 180,E1 -21874.188,E2 -21874.188} C_VEL
LIN {X 0,Y 191.048,Z 452.74,A -85,B 0,C 180,E1 -21878.461,E2 -21878.461} C_VEL
LIN {X 0,Y 190.124,Z 456.779,A -85,B 0,C 180,E1 -21882.813,E2 -21882.813} C_VEL
LIN {X 0,Y 189.768,Z 459.518,A -85,B 0,C 180,E1 -21887.233,E2 -21887.233} C_VEL
LIN {X 0,Y 189.901,Z 461.003,A -85,B 0,C 180,E1 -21891.72,E2 -21891.72} C_VEL
LIN {X 0,Y 190.452,Z 461.236,A -85,B 0,C 180,E1 -21896.283,E2 -21896.283} C_VEL
LIN {X 0,Y 191.76,Z 460.169,A -85,B 0,C 180,E1 -21900.87,E2 -21900.87} C_VEL
LIN {X 0,Y 193.968,Z 457.751,A -85,B 0,C 180,E1 -21905.43,E2 -21905.43} C_VEL
LIN {X 0,Y 197.182,Z 453.898,A -85,B 0,C 180,E1 -21909.907,E2 -21909.907} C_VEL
LIN {X 0,Y 201.363,Z 448.497,A -85,B 0,C 180,E1 -21914.269,E2 -21914.269} C_VEL
LIN {X 0,Y 205.236,Z 443.361,A -85,B 0,C 180,E1 -21917.409,E2 -21917.409} C_VEL
LIN {X 0,Y 210.412,Z 436.001,A -85,B 0,C 180,E1 -21920.947,E2 -21920.947} C_VEL
LIN {X 0,Y 216.187,Z 427.284,A -85,B 0,C 180,E1 -21924.185,E2 -21924.185} C_VEL
LIN {X 0,Y 222.079,Z 417.646,A -85,B 0,C 180,E1 -21926.994,E2 -21926.994} C_VEL
LIN {X 0,Y 228.189,Z 406.448,A -85,B 0,C 180,E1 -21929.583,E2 -21929.583} C_VEL
LIN {X 0,Y 233.647,Z 395.345,A -85,B 0,C 180,E1 -21931.621,E2 -21931.621} C_VEL
LIN {X 0,Y 239.055,Z 382.816,A -85,B 0,C 180,E1 -21933.451,E2 -21933.451} C_VEL
LIN {X 0,Y 244.083,Z 368.823,A -85,B 0,C 180,E1 -21935.092,E2 -21935.092} C_VEL
LIN {X 0,Y 248.336,Z 354.812,A -85,B 0,C 180,E1 -21936.334,E2 -21936.334} C_VEL
LIN {X 0,Y 251.969,Z 339.367,A -85,B 0,C 180,E1 -21937.377,E2 -21937.377} C_VEL
LIN {X 0,Y 254.526,Z 324.991,A -85,B 0,C 180,E1 -21938.061,E2 -21938.061} C_VEL
LIN {X 0,Y 256.219,Z 309.608,A -85,B 0,C 180,E1 -21938.574,E2 -21938.574} C_VEL
LIN {X 0,Y 261.025,Z 248.227,A -85,B 0,C 180,E1 -21940.119,E2 -21940.119} C_VEL
LIN {X 0,Y 256.39,Z 238.831,A -85,B 0,C 180,E1 -21942.399,E2 -21942.399} C_VEL
LIN {X 0,Y 251.367,Z 230.377,A -85,B 0,C 180,E1 -21945.125,E2 -21945.125} C_VEL
LIN {X 0,Y 246.23,Z 222.458,A -85,B 0,C 180,E1 -21948.3,E2 -21948.3} C_VEL
LIN {X 0,Y 243.143,Z 218.043,A -85,B 0,C 180,E1 -21950.484,E2 -21950.484} C_VEL
LIN {X 0,Y 240.192,Z 213.702,A -85,B 0,C 180,E1 -21952.961,E2 -21952.961} C_VEL
LIN {X 0,Y 237.365,Z 209.556,A -85,B 0,C 180,E1 -21955.784,E2 -21955.784} C_VEL
LIN {X 0,Y 235.013,Z 207.069,A -85,B 0,C 180,E1 -21958.557,E2 -21958.557} C_VEL
LIN {X 0,Y 233.837,Z 204.404,A -85,B 0,C 180,E1 -21960.571,E2 -21960.571} C_VEL
LIN {X 0,Y 231.201,Z 202.27,A -85,B 0,C 180,E1 -21968.742,E2 -21968.742} C_VEL
LIN {X 0,Y 232.225,Z 203.7,A -85,B 0,C 180,E1 -21974.926,E2 -21974.926} C_VEL
LIN {X 0,Y 233.775,Z 204.908,A -85,B 0,C 180,E1 -21978.101,E2 -21978.101} C_VEL
LIN {X 0,Y 235.462,Z 208.05,A -85,B 0,C 180,E1 -21980.761,E2 -21980.761} C_VEL
LIN {X 0,Y 237.191,Z 210.004,A -85,B 0,C 180,E1 -21982.77,E2 -21982.77} C_VEL
LIN {X 0,Y 238.544,Z 212.168,A -85,B 0,C 180,E1 -21984.222,E2 -21984.222} C_VEL
LIN {X 0,Y 241.506,Z 217.038,A -85,B 0,C 180,E1 -21986.986,E2 -21986.986} C_VEL
LIN {X 0,Y 244.799,Z 222.544,A -85,B 0,C 180,E1 -21989.554,E2 -21989.554} C_VEL
LIN {X 0,Y 248.88,Z 229.785,A -85,B 0,C 180,E1 -21992.29,E2 -21992.29} C_VEL
LIN {X 0,Y 250.256,Z 232.329,A -85,B 0,C 180,E1 -21993.139,E2 -21993.139} C_VEL
LIN {X 0,Y 251.714,Z 236.285,A -85,B 0,C 180,E1 -21994.082,E2 -21994.082} C_VEL
LIN {X 0,Y 253.402,Z 244.337,A -85,B 0,C 180,E1 -21995.341,E2 -21995.341} C_VEL
LIN {X 0,Y 254.667,Z 251.089,A -85,B 0,C 180,E1 -21996.283,E2 -21996.283} C_VEL
LIN {X 0,Y 255.963,Z 255.756,A -85,B 0,C 180,E1 -21997.075,E2 -21997.075} C_VEL
LIN {X 0,Y 256.52,Z 257.154,A -85,B 0,C 180,E1 -21997.368,E2 -21997.368} C_VEL
LIN {X 0,Y 256.707,Z 257.593,A -85,B 0,C 180,E1 -21997.463,E2 -21997.463} C_VEL
LIN {X 0,Y 251.141,Z 325.255,A -85,B 0,C 180,E1 -21999.212,E2 -21999.212} C_VEL
LIN {X 0,Y 248.69,Z 340.781,A -85,B 0,C 180,E1 -21999.797,E2 -21999.797} C_VEL
LIN {X 0,Y 245.29,Z 355.752,A -85,B 0,C 180,E1 -22000.601,E2 -22000.601} C_VEL
LIN {X 0,Y 241.028,Z 370.229,A -85,B 0,C 180,E1 -22001.654,E2 -22001.654} C_VEL
LIN {X 0,Y 236.418,Z 383.365,A -85,B 0,C 180,E1 -22002.944,E2 -22002.944} C_VEL
LIN {X 0,Y 230.943,Z 396.361,A -85,B 0,C 180,E1 -22004.538,E2 -22004.538} C_VEL
LIN {X 0,Y 225.44,Z 408.02,A -85,B 0,C 180,E1 -22006.391,E2 -22006.391} C_VEL
LIN {X 0,Y 219.852,Z 418.508,A -85,B 0,C 180,E1 -22008.448,E2 -22008.448} C_VEL
LIN {X 0,Y 214.069,Z 428.276,A -85,B 0,C 180,E1 -22010.804,E2 -22010.804} C_VEL
LIN {X 0,Y 207.8,Z 437.887,A -85,B 0,C 180,E1 -22013.711,E2 -22013.711} C_VEL
LIN {X 0,Y 202.238,Z 445.944,A -85,B 0,C 180,E1 -22016.817,E2 -22016.817} C_VEL
LIN {X 0,Y 197.404,Z 452.619,A -85,B 0,C 180,E1 -22020.105,E2 -22020.105} C_VEL
LIN {X 0,Y 192.662,Z 458.851,A -85,B 0,C 180,E1 -22024.041,E2 -22024.041} C_VEL
LIN {X 0,Y 188.832,Z 463.735,A -85,B 0,C 180,E1 -22028.15,E2 -22028.15} C_VEL
LIN {X 0,Y 186.047,Z 467.395,A -85,B 0,C 180,E1 -22032.411,E2 -22032.411} C_VEL
LIN {X 0,Y 184.186,Z 469.902,A -85,B 0,C 180,E1 -22036.766,E2 -22036.766} C_VEL
LIN {X 0,Y 183.262,Z 471.256,A -85,B 0,C 180,E1 -22041.177,E2 -22041.177} C_VEL
LIN {X 0,Y 182.977,Z 471.466,A -85,B 0,C 180,E1 -22045.595,E2 -22045.595} C_VEL
LIN {X 0,Y 183.216,Z 470.559,A -85,B 0,C 180,E1 -22050.001,E2 -22050.001} C_VEL
LIN {X 0,Y 183.113,Z 468.458,A -85,B 0,C 180,E1 -22054.403,E2 -22054.403} C_VEL
LIN {X 0,Y 183.278,Z 465.109,A -85,B 0,C 180,E1 -22058.824,E2 -22058.824} C_VEL
LIN {X 0,Y 184.011,Z 460.405,A -85,B 0,C 180,E1 -22063.249,E2 -22063.249} C_VEL
LIN {X 0,Y 185.586,Z 454.237,A -85,B 0,C 180,E1 -22067.636,E2 -22067.636} C_VEL
LIN {X 0,Y 188.037,Z 446.45,A -85,B 0,C 180,E1 -22071.949,E2 -22071.949} C_VEL
LIN {X 0,Y 190.919,Z 438.083,A -85,B 0,C 180,E1 -22075.629,E2 -22075.629} C_VEL
LIN {X 0,Y 194.552,Z 428.015,A -85,B 0,C 180,E1 -22079.189,E2 -22079.189} C_VEL
LIN {X 0,Y 198.139,Z 417.652,A -85,B 0,C 180,E1 -22082.145,E2 -22082.145} C_VEL
LIN {X 0,Y 201.873,Z 406.397,A -85,B 0,C 180,E1 -22084.757,E2 -22084.757} C_VEL
LIN {X 0,Y 205.275,Z 395.537,A -85,B 0,C 180,E1 -22086.81,E2 -22086.81} C_VEL
LIN {X 0,Y 208.931,Z 382.605,A -85,B 0,C 180,E1 -22088.794,E2 -22088.794} C_VEL
LIN {X 0,Y 212.353,Z 368.533,A -85,B 0,C 180,E1 -22090.495,E2 -22090.495} C_VEL
LIN {X 0,Y 215.068,Z 355.182,A -85,B 0,C 180,E1 -22091.746,E2 -22091.746} C_VEL
LIN {X 0,Y 217.553,Z 339.829,A -85,B 0,C 180,E1 -22092.799,E2 -22092.799} C_VEL
LIN {X 0,Y 219.18,Z 325.014,A -85,B 0,C 180,E1 -22093.504,E2 -22093.504} C_VEL
LIN {X 0,Y 224.525,Z 236.871,A -85,B 0,C 180,E1 -22096.139,E2 -22096.139} C_VEL
LIN {X 0,Y 224.156,Z 234.988,A -85,B 0,C 180,E1 -22096.296,E2 -22096.296} C_VEL
LIN {X 0,Y 217.533,Z 217.983,A -85,B 0,C 180,E1 -22098.485,E2 -22098.485} C_VEL
LIN {X 0,Y 210.972,Z 203.714,A -85,B 0,C 180,E1 -22100.734,E2 -22100.734} C_VEL
LIN {X 0,Y 204.903,Z 191.859,A -85,B 0,C 180,E1 -22102.96,E2 -22102.96} C_VEL
LIN {X 0,Y 200.762,Z 184.88,A -85,B 0,C 180,E1 -22104.553,E2 -22104.553} C_VEL
LIN {X 0,Y 195.324,Z 177.116,A -85,B 0,C 180,E1 -22106.732,E2 -22106.732} C_VEL
LIN {X 0,Y 192.724,Z 173.396,A -85,B 0,C 180,E1 -22107.846,E2 -22107.846} C_VEL
LIN {X 0,Y 189.887,Z 169.778,A -85,B 0,C 180,E1 -22109.101,E2 -22109.101} C_VEL
LIN {X 0,Y 188.958,Z 168.196,A -85,B 0,C 180,E1 -22109.553,E2 -22109.553} C_VEL
LIN {X 0,Y 186.715,Z 166.106,A -85,B 0,C 180,E1 -22110.562,E2 -22110.562} C_VEL
LIN {X 0,Y 185.682,Z 163.564,A -85,B 0,C 180,E1 -22111.147,E2 -22111.147} C_VEL
LIN {X 0,Y 185.584,Z 162.957,A -85,B 0,C 180,E1 -22111.285,E2 -22111.285} C_VEL
LIN {X 0,Y 185.583,Z 162.983,A -85,B 0,C 180,E1 -22115.383,E2 -22115.383} C_VEL
LIN {X 0,Y 185.676,Z 162.979,A -85,B 0,C 180,E1 -22121.137,E2 -22121.137} C_VEL
LIN {X 0,Y 185.686,Z 162.976,A -85,B 0,C 180,E1 -22124.637,E2 -22124.637} C_VEL
LIN {X 0,Y 185.892,Z 162.953,A -85,B 0,C 180,E1 -22129.42,E2 -22129.42} C_VEL
LIN {X 0,Y 185.934,Z 162.943,A -85,B 0,C 180,E1 -22133.49,E2 -22133.49} C_VEL
LIN {X 0,Y 186.181,Z 162.878,A -85,B 0,C 180,E1 -22137.838,E2 -22137.838} C_VEL
LIN {X 0,Y 186.383,Z 162.843,A -85,B 0,C 180,E1 -22140.001,E2 -22140.001} C_VEL
LIN {X 0,Y 185.885,Z 162.955,A -85,B 0,C 180,E1 -22144.338,E2 -22144.338} C_VEL
LIN {X 0,Y 185.976,Z 162.893,A -85,B 0,C 180,E1 -22148.695,E2 -22148.695} C_VEL
LIN {X 0,Y 185.707,Z 162.965,A -85,B 0,C 180,E1 -22153.125,E2 -22153.125} C_VEL
LIN {X 0,Y 185.629,Z 162.984,A -85,B 0,C 180,E1 -22158.821,E2 -22158.821} C_VEL
LIN {X 0,Y 185.566,Z 162.996,A -85,B 0,C 180,E1 -22164.635,E2 -22164.635} C_VEL
LIN {X 0,Y 185.548,Z 162.949,A -85,B 0,C 180,E1 -22169.5,E2 -22169.5} C_VEL
LIN {X 0,Y 185.501,Z 163,A -85,B 0,C 180,E1 -22174.633,E2 -22174.633} C_VEL
LIN {X 0,Y 185.504,Z 162.964,A -85,B 0,C 180,E1 -22177.315,E2 -22177.315} C_VEL
LIN {X 0,Y 185.467,Z 162.987,A -85,B 0,C 180,E1 -22180.722,E2 -22180.722} C_VEL
LIN {X 0,Y 185.459,Z 162.976,A -85,B 0,C 180,E1 -22186.057,E2 -22186.057} C_VEL
LIN {X 0,Y 185.455,Z 162.996,A -85,B 0,C 180,E1 -22188.184,E2 -22188.184} C_VEL
LIN {X 0,Y 186.331,Z 165.621,A -85,B 0,C 180,E1 -22188.736,E2 -22188.736} C_VEL
LIN {X 0,Y 188.222,Z 167.792,A -85,B 0,C 180,E1 -22189.623,E2 -22189.623} C_VEL
LIN {X 0,Y 189.237,Z 168.66,A -85,B 0,C 180,E1 -22190.066,E2 -22190.066} C_VEL
LIN {X 0,Y 191.181,Z 171.8,A -85,B 0,C 180,E1 -22190.979,E2 -22190.979} C_VEL
LIN {X 0,Y 192.918,Z 173.764,A -85,B 0,C 180,E1 -22191.716,E2 -22191.716} C_VEL
LIN {X 0,Y 195.778,Z 177.57,A -85,B 0,C 180,E1 -22192.92,E2 -22192.92} C_VEL
LIN {X 0,Y 202.163,Z 186.978,A -85,B 0,C 180,E1 -22195.461,E2 -22195.461} C_VEL
LIN {X 0,Y 209.452,Z 198.542,A -85,B 0,C 180,E1 -22198.1,E2 -22198.1} C_VEL
LIN {X 0,Y 217.379,Z 212.672,A -85,B 0,C 180,E1 -22200.72,E2 -22200.72} C_VEL
LIN {X 0,Y 222.656,Z 223.058,A -85,B 0,C 180,E1 -22202.349,E2 -22202.349} C_VEL
LIN {X 0,Y 224.864,Z 228.822,A -85,B 0,C 180,E1 -22203.067,E2 -22203.067} C_VEL
LIN {X 0,Y 219.421,Z 315.929,A -85,B 0,C 180,E1 -22205.644,E2 -22205.644} C_VEL
LIN {X 0,Y 217.717,Z 331.915,A -85,B 0,C 180,E1 -22206.454,E2 -22206.454} C_VEL
LIN {X 0,Y 215.334,Z 347.138,A -85,B 0,C 180,E1 -22207.575,E2 -22207.575} C_VEL
LIN {X 0,Y 212.592,Z 360.849,A -85,B 0,C 180,E1 -22208.929,E2 -22208.929} C_VEL
LIN {X 0,Y 209.169,Z 375.346,A -85,B 0,C 180,E1 -22210.792,E2 -22210.792} C_VEL
LIN {X 0,Y 205.578,Z 388.087,A -85,B 0,C 180,E1 -22212.85,E2 -22212.85} C_VEL
LIN {X 0,Y 201.64,Z 400.549,A -85,B 0,C 180,E1 -22215.362,E2 -22215.362} C_VEL
LIN {X 0,Y 197.81,Z 411.875,A -85,B 0,C 180,E1 -22218.211,E2 -22218.211} C_VEL
LIN {X 0,Y 193.88,Z 422.896,A -85,B 0,C 180,E1 -22221.662,E2 -22221.662} C_VEL
LIN {X 0,Y 190.692,Z 431.911,A -85,B 0,C 180,E1 -22225.195,E2 -22225.195} C_VEL
LIN {X 0,Y 187.955,Z 439.604,A -85,B 0,C 180,E1 -22228.928,E2 -22228.928} C_VEL
LIN {X 0,Y 185.663,Z 446.694,A -85,B 0,C 180,E1 -22233.254,E2 -22233.254} C_VEL
LIN {X 0,Y 184.22,Z 451.818,A -85,B 0,C 180,E1 -22237.288,E2 -22237.288} C_VEL
LIN {X 0,Y 183.301,Z 455.536,A -85,B 0,C 180,E1 -22241.052,E2 -22241.052} C_VEL
LIN {X 0,Y 182.776,Z 458.785,A -85,B 0,C 180,E1 -22245.613,E2 -22245.613} C_VEL
LIN {X 0,Y 182.677,Z 460.79,A -85,B 0,C 180,E1 -22250.257,E2 -22250.257} C_VEL
LIN {X 0,Y 183.108,Z 461.529,A -85,B 0,C 180,E1 -22254.973,E2 -22254.973} C_VEL
LIN {X 0,Y 184.232,Z 460.966,A -85,B 0,C 180,E1 -22259.729,E2 -22259.729} C_VEL
LIN {X 0,Y 186.266,Z 459.076,A -85,B 0,C 180,E1 -22264.468,E2 -22264.468} C_VEL
LIN {X 0,Y 189.294,Z 455.796,A -85,B 0,C 180,E1 -22269.135,E2 -22269.135} C_VEL
LIN {X 0,Y 193.355,Z 451.031,A -85,B 0,C 180,E1 -22273.677,E2 -22273.677} C_VEL
LIN {X 0,Y 198.549,Z 444.652,A -85,B 0,C 180,E1 -22278.015,E2 -22278.015} C_VEL
LIN {X 0,Y 203.899,Z 437.515,A -85,B 0,C 180,E1 -22281.652,E2 -22281.652} C_VEL
LIN {X 0,Y 209.536,Z 429.501,A -85,B 0,C 180,E1 -22284.814,E2 -22284.814} C_VEL
LIN {X 0,Y 215.872,Z 419.751,A -85,B 0,C 180,E1 -22287.828,E2 -22287.828} C_VEL
LIN {X 0,Y 222.165,Z 408.961,A -85,B 0,C 180,E1 -22290.45,E2 -22290.45} C_VEL
LIN {X 0,Y 227.836,Z 398.084,A -85,B 0,C 180,E1 -22292.544,E2 -22292.544} C_VEL
LIN {X 0,Y 233.617,Z 385.447,A -85,B 0,C 180,E1 -22294.488,E2 -22294.488} C_VEL
LIN {X 0,Y 238.457,Z 373.046,A -85,B 0,C 180,E1 -22296.015,E2 -22296.015} C_VEL
LIN {X 0,Y 243.143,Z 358.741,A -85,B 0,C 180,E1 -22297.389,E2 -22297.389} C_VEL
LIN {X 0,Y 246.935,Z 344.155,A -85,B 0,C 180,E1 -22298.463,E2 -22298.463} C_VEL
LIN {X 0,Y 250.087,Z 328.433,A -85,B 0,C 180,E1 -22299.272,E2 -22299.272} C_VEL
LIN {X 0,Y 252.108,Z 312.78,A -85,B 0,C 180,E1 -22299.828,E2 -22299.828} C_VEL
LIN {X 0,Y 257.092,Z 251.557,A -85,B 0,C 180,E1 -22301.385,E2 -22301.385} C_VEL
LIN {X 0,Y 253.601,Z 244.21,A -85,B 0,C 180,E1 -22303.241,E2 -22303.241} C_VEL
LIN {X 0,Y 248.828,Z 236.004,A -85,B 0,C 180,E1 -22305.963,E2 -22305.963} C_VEL
LIN {X 0,Y 244.053,Z 228.459,A -85,B 0,C 180,E1 -22309.07,E2 -22309.07} C_VEL
LIN {X 0,Y 241.167,Z 224.201,A -85,B 0,C 180,E1 -22311.251,E2 -22311.251} C_VEL
LIN {X 0,Y 238.547,Z 220.154,A -85,B 0,C 180,E1 -22313.579,E2 -22313.579} C_VEL
LIN {X 0,Y 236.124,Z 216.427,A -85,B 0,C 180,E1 -22316.11,E2 -22316.11} C_VEL
LIN {X 0,Y 233.83,Z 213.927,A -85,B 0,C 180,E1 -22318.912,E2 -22318.912} C_VEL
LIN {X 0,Y 232.632,Z 211.3,A -85,B 0,C 180,E1 -22321.08,E2 -22321.08} C_VEL
LIN {X 0,Y 230.305,Z 209.316,A -85,B 0,C 180,E1 -22328.776,E2 -22328.776} C_VEL
LIN {X 0,Y 231.704,Z 211.062,A -85,B 0,C 180,E1 -22335.841,E2 -22335.841} C_VEL
LIN {X 0,Y 232.679,Z 211.882,A -85,B 0,C 180,E1 -22337.783,E2 -22337.783} C_VEL
LIN {X 0,Y 234.434,Z 215.088,A -85,B 0,C 180,E1 -22340.628,E2 -22340.628} C_VEL
LIN {X 0,Y 236.199,Z 217.233,A -85,B 0,C 180,E1 -22342.723,E2 -22342.723} C_VEL
LIN {X 0,Y 237.135,Z 218.923,A -85,B 0,C 180,E1 -22343.772,E2 -22343.772} C_VEL
